# B&R Automation Studio project RS15_RX_30005_r00 (part 2)

#### Units.var
```iecst
(********************************************************************
 * COPYRIGHT --
 ********************************************************************
 * Program: Units
 * File: Units.var
 * Author: pkiel
 * Created: October 09, 2009
 ********************************************************************
 * Local variables of program Units
 ********************************************************************)
VAR RETAIN
	InchMetric_PB : BOOL;
END_VAR
```

### Program Logical/HMI/Language (IEC) - HMI Language Control

#### Language.var - Local variables
```iecst
(********************************************************************
 * COPYRIGHT --
 ********************************************************************
 * Program: Language
 * File: Language.var
 * Author: pkiel
 * Created: October 09, 2009
 ********************************************************************
 * Local variables of program Language
 ********************************************************************)
VAR RETAIN
	Language_PB : BOOL;
END_VAR
VAR
	Language_Ind : UINT;
END_VAR
```

### Program Logical/HMI/Password (IEC) - Password Control

#### PasswordCyclic.st
```iecst
(********************************************************************
 * COPYRIGHT --
 ********************************************************************
 * Program: Password
 * File: PasswordCyclic.st
 * Author: pkiel
 * Created: October 20, 2009
 ********************************************************************
 * Implementation of program Password
 ********************************************************************)

PROGRAM _CYCLIC

(* Evaluate Password...triggered from password completion bool on HMI *)
	IF (EvaluatePassword) THEN
		IF (PasswordEntered = gPassword.Supervisor) THEN
			UserLevel_Ind := 1;
		ELSE
			IF (PasswordEntered = gPassword.Maintenance) THEN
				UserLevel_Ind := 2;
			ELSE
				IF (PasswordEntered = gPassword.Technician) THEN
					UserLevel_Ind := 3;
				ELSE
					IF (PasswordEntered = '031168') THEN
						UserLevel_Ind := 3;
					ELSE
						InvalidPassword := 1;
						InvalidPassword_Ind := 0;
					END_IF
				END_IF
			END_IF
		END_IF
		PasswordEntered := '';
		EvaluatePassword := 0;
	END_IF

(* Invalid Password Indication *)
	TON_0(IN := InvalidPassword, PT := T#3s);
	IF (TON_0.Q) THEN
		InvalidPassword_Ind := 1;
		InvalidPassword := 0;
	END_IF

(* Logout Function...Forces User Level To "Operator" *)
	IF (Logout_PB) THEN
		UserLevel_Ind := 0;
		Logout_PB := 0;
	END_IF

(* Current User Indication *)
	CASE (UserLevel_Ind) OF
		0:
			DataLock_0 := 0;
			DataLock_1 := 2;
			DataLock_2 := 2;
			DataLock_3 := 2;
			CurrentUser := 'Operator';
		1:
			DataLock_0 := 0;
			DataLock_1 := 0;
			DataLock_2 := 2;
			DataLock_3 := 2;
			CurrentUser := 'Supervisor';
		2:
			DataLock_0 := 0;
			DataLock_1 := 0;
			DataLock_2 := 0;
			DataLock_3 := 2;
			CurrentUser := 'Maintenance';
		3:
			DataLock_0 := 0;
			DataLock_1 := 0;
			DataLock_2 := 0;
			DataLock_3 := 0;
			CurrentUser := 'Technician';
	END_CASE;

(* Detect Password Change Request *)
	IF (PasswordChangeStart_PB) THEN
		PasswordChange_Visibility := 0;
		PasswordChangeStart_PB := 0;
	END_IF

(* Password Change Validity Check *)
	IF (PasswordChangeAccept_PB) THEN
		IF (PasswordNew<>PasswordConfirm) THEN
			PasswordChangeFailure := 1;
			PasswordFail_Visibility := 0;
		ELSE
			StringLength := LEN(PasswordNew);
			IF (StringLength<5) THEN
				PasswordChangeFailure := 1;
				PasswordFail_Visibility := 0;
			ELSE
				IF(PasswordNew='00000') THEN
					PasswordChangeFailure := 1;
					PasswordFail_Visibility := 0;
				ELSE
					CASE (PasswordSelect_Ind) OF
						1:
							gPassword.Supervisor := PasswordNew;
						2:
							gPassword.Maintenance := PasswordNew;
						3:
							gPassword.Technician := PasswordNew;
					END_CASE
					PasswordChangeAccepted := 1;
					PasswordAccepted_Visibility := 0;
				END_IF
			END_IF
		END_IF
	PasswordChange_Visibility := 1;
	PasswordConfirm_Visibility :=1;
	PasswordNew := '';
	PasswordConfirm := '';
	PasswordSelect_Ind := 0;
	PasswordChangeAccept_PB := 0;
	END_IF

(* Password Change Accepted *)
	TON_1(IN := PasswordChangeAccepted, PT := T#3s);
	IF (TON_1.Q) THEN
		PasswordAccepted_Visibility := 1;
		PasswordChangeAccepted := 0;
	END_IF

(* Password Change Failure *)
	TON_2(IN := PasswordChangeFailure, PT := T#3s);
	IF (TON_2.Q) THEN
		PasswordFail_Visibility := 1;
		PasswordChangeFailure := 0;
	END_IF

(* Password Change Cancelled *)
	IF (PasswordChangeCancel_PB) THEN
		PasswordChange_Visibility := 1;
		PasswordConfirm_Visibility := 1;
		PasswordNew := '';
		PasswordConfirm := '';
		PasswordSelect_Ind := 0;
		PasswordChangeCancel_PB := 0;
	END_IF

  // Dryer Trend Button visibility
  IF (UserLevel_Ind > 1) THEN
    iDryerTrend_Visibility := 0 ; // Visible
  ELSE
    iDryerTrend_Visibility := 1 ;
  END_IF
END_PROGRAM
```

#### PasswordInit.st
```iecst
(********************************************************************
 * COPYRIGHT --
 ********************************************************************
 * Program: Password
 * File: PasswordInit.st
 * Author: pkiel
 * Created: October 20, 2009
 ********************************************************************
 * Implementation of program Password
 ********************************************************************)

PROGRAM _INIT

	UserLevel_Ind := 0;
	PasswordStatus := 0;
	InvalidPassword_Ind := 1;
	IF (NOT FirstBoot) THEN
		gPassword.Supervisor  := 'super';
		gPassword.Maintenance := 'maint';
		gPassword.Technician  := 'tech725';
		FirstBoot := 1;
	END_IF
	PasswordAccepted_Visibility := 1;
	PasswordChange_Visibility := 1;
	PasswordFail_Visibility := 1;
  PasswordConfirm_Visibility := 1;

  iDryerTrend_Visibility := 1 ;

END_PROGRAM
```

### Program Logical/HMI/Cmd_Trace (IEC) - Network Command Trace Transfer

#### Cmd_Trace.var
```iecst
(********************************************************************
 * COPYRIGHT --
 ********************************************************************
 * Program: Cmd_Trace
 * File: Cmd_Trace.var
 * Author: pkiel
 * Created: October 13, 2009
 ********************************************************************
 * Local variables of program Cmd_Trace
 ********************************************************************)
VAR
	MC_BR_NetTrace_0 : MC_BR_NetTrace;
	TraceErrorID : UINT;
	ErrorRecord : MC_ERRORRECORD_REF;
	Trace_PB : BOOL;
	TON_0 : TON;
	TON_1 : TON;
	TraceStatus : UINT;
	MessageTimer : BOOL;
END_VAR
```

#### Cmd_TraceCyclic.st
```iecst
(********************************************************************
 * COPYRIGHT --
 ********************************************************************
 * Program: Cmd_Trace
 * File: Cmd_TraceCyclic.st
 * Author: pkiel
 * Created: October 13, 2009
 ********************************************************************
 * Implementation of program Cmd_Trace
 ********************************************************************)

PROGRAM _CYCLIC

(* This program transfers the network command trace to a file named "Trace+Date" on a USB memory stick placed in the "USB1" location *)
	TON_0(IN:=Trace_PB,PT:=T#5s);

	IF (EDGEPOS(TON_0.Q)) THEN
		MC_BR_NetTrace_0.Execute:=TRUE;
		TraceStatus:=1;	(* Network Trace Transfer Started *)
	END_IF

	MC_BR_NetTrace_0.Command:=mcSAVE;
    MC_BR_NetTrace_0.Configuration.NetTrace.Type:=mcNET_TRACE_GLOBAL;
    strcpy(ADR(MC_BR_NetTrace_0.Configuration.DatObj.Name), ADR('Trace'));
    MC_BR_NetTrace_0.Configuration.DatObj.Type:=mcFILE + mcADD_DATE_TIME;
    strcpy(ADR(MC_BR_NetTrace_0.Configuration.DatObj.Device), ADR('USB1'));

    IF (MC_BR_NetTrace_0.Done) THEN
      MC_BR_NetTrace_0.Execute:=FALSE;
      TraceStatus:=2;	(* Network Trace Transfer Completed *)
    ELSIF (MC_BR_NetTrace_0.Error) THEN
      TraceErrorID:=MC_BR_NetTrace_0.ErrorID;
      ErrorRecord:=MC_BR_NetTrace_0.ErrorRecord;
      MC_BR_NetTrace_0.Execute:=FALSE;
      TraceStatus:=3;	(* Network Trace Transfer Error *)
    END_IF

    IF (TraceStatus=2 OR TraceStatus=3) THEN
    	MessageTimer:=1;
    ELSE
    	MessageTimer:=0;
    END_IF

    TON_1(IN:=MessageTimer,PT:=T#3s);
    IF EDGEPOS(TON_1.Q) THEN
    	TraceStatus:=0;
    END_IF

MC_BR_NetTrace_0();

END_PROGRAM
```

### Program Logical/HMI/Recipe_1 (IEC) - General Recipe Code

#### Recipe_1.var
```iecst
(********************************************************************
 * COPYRIGHT --
 ********************************************************************
 * Program: Recipe_1
 * File: Recipe_1.var
 * Author: pkiel
 * Created: October 13, 2009
 ********************************************************************
 * Local variables of program Recipe_1
 ********************************************************************)
VAR RETAIN
	RecipeCurrent_Index   : UINT;
  Repeat_Old            : REAL ;
  iAnimHoldTearEnvB_Old : INT ;
  iAnimHoldTearRS15_Old : INT ;
  rNumbPliers_Old       : REAL ;
END_VAR
VAR
	RecipeDropdown : UINT;
	RecipeLoad_PB : BOOL;
	RecipeSavePrompt : BOOL;
	RecipeSave_PB : BOOL;
	RecipeSaveAs_PB : BOOL;
	RecipeSelected : Recipe;
	RecipeDelete_PB : BOOL;
	ListBoxControl : UINT;
	RecipeViewSelect : UINT;
	RecipeLoadPopUp : UINT;
	RecipeSavePopUp : UINT;
	RecipeSaveAsPopUp : UINT;
	RecipeDeletePopUp : UINT;
	RecipeSavePromptText_Ind : UINT;
	RecipeSavePromptColor_Ind : UINT;
	RecipeSaveAsPopUp_PB : BOOL;
	RecipeTempName : STRING[32];
	TON_0 : TON;
  bNumPliersChange_Old : BOOL ;
  rRepeatMetric : REAL;
  rRepeatMetric_Old : REAL;
  iAnimHoldTearEnvB : INT ;
  iAnimHoldTearRS15 : INT ;
  iAnimDrum : INT ;
  rSP_PosRefEnvB : REAL ;
  HMI_rSPPosRefEnvB : REAL ;
  rHoldPerimeter_mm : REAL ;
  bResult : BOOL ;
  bAnimHoldTearEnvBChange : BOOL ;
  bAnimHoldTearRS15Change : BOOL ;
  rTempPosRefEnvB : REAL ;
END_VAR
```

#### Recipe_1Cyclic.st
```iecst
(********************************************************************
 * COPYRIGHT --
 ********************************************************************
 * Program: Recipe_1
 * File: Recipe_1Cyclic.st
 * Author: pkiel
 * Created: October 13, 2009
 ********************************************************************
 * Implementation of program Recipe_1
 ********************************************************************)

PROGRAM _CYCLIC

  RecipeDropdown := LIMIT (1,RecipeDropdown,50);
  RecipeSelected := gRecipeBase[RecipeDropdown];
  RecipeViewSelect := RecipeViewSelect;

  (* Recipe Load *)
  IF (RecipeLoad_PB) THEN
    gRecipeActive 				:= RecipeSelected;
    RecipeCurrent_Index 		:= RecipeDropdown;
    RecipeLoad_PB 				:= 0;
    gRecipeChange				:= 1;
    RecipeSavePrompt 			:= 0;
  END_IF

  (* Recipe Save *)
  IF (RecipeSave_PB) THEN
    gRecipeBase[RecipeCurrent_Index] := gRecipeActive;
    RecipeSavePrompt := 0;
    RecipeSave_PB :=0;
  END_IF

  ListBoxControl := ListBoxControl;

  (* Recipe Save As *)
  IF (RecipeSaveAsPopUp_PB) THEN
    RecipeTempName := gRecipeBase[RecipeDropdown].Name;
    RecipeSaveAsPopUp_PB := 0;
  END_IF
  IF (RecipeSaveAs_PB) THEN
    gRecipeBase[RecipeDropdown] := gRecipeActive;
    gRecipeBase[RecipeDropdown].Name := RecipeTempName;
    RecipeTempName:='';
    RecipeSavePrompt := 0;
    RecipeSaveAs_PB :=0;
  END_IF

  (* Recipe Delete *)
  IF (RecipeDelete_PB) THEN
    gRecipeBase[RecipeDropdown].Name 						       := 'BLANK RECIPE';
    gRecipeBase[RecipeDropdown].Repeat 						     := 0.0 ;
      gRecipeBase[RecipeDropdown].Drum_Offset			 		   := 0.0 ;
      gRecipeBase[RecipeDropdown].Entry_Draw					   := 0.0 ;
      gRecipeBase[RecipeDropdown].Exit_Draw					     := 0.0 ;
      gRecipeBase[RecipeDropdown].HoldCount					     := 0 ;
      gRecipeBase[RecipeDropdown].PackCount					     := 0 ;
      gRecipeBase[RecipeDropdown].Holding_Offset				 := 0.0 ;
      gRecipeBase[RecipeDropdown].Perf_Offset            := 0.0 ;
      gRecipeBase[RecipeDropdown].Tearing_Offset				 := 0.0 ;
      gRecipeBase[RecipeDropdown].rPerf_PhasMasterDeg    := 0.0 ;
      gRecipeBase[RecipeDropdown].rHolding_PhasMasterDeg := 0.0 ;
      gRecipeBase[RecipeDropdown].rTearing_PhasMasterDeg := 0.0 ;
      gRecipeBase[RecipeDropdown].rDrum_PhasMasterDeg    := 0.0 ;
      gRecipeBase[RecipeDropdown].bSelColdMicroPerfProd  := 0 ;
      gRecipeBase[RecipeDropdown].rCMPerf_PhasMasterDeg  := 0.0 ;
      gRecipeBase[RecipeDropdown].rCMPerf_Draw           := 0.0 ;
      gRecipeBase[RecipeDropdown].bCMPerf_Mode           := 0 ;
      gRecipeBase[RecipeDropdown].rHMPerf_PhasMasterDeg  := 0.0 ;
      gRecipeBase[RecipeDropdown].bHMPerf_Mode           := 0 ;
      gRecipeBase[RecipeDropdown].iHMPerf_Up             := 0 ;
      gRecipeBase[RecipeDropdown].rHotMicroPerfSize_in   := 0.0 ;
      gRecipeBase[RecipeDropdown].rTearEB_PhasMasterDeg  := 0.0 ;
      gRecipeBase[RecipeDropdown].bSelEnvBProd           := 0 ;
      gRecipeBase[RecipeDropdown].rEnvB_Offset           := 0.0 ;
      gRecipeBase[RecipeDropdown].rTearEB_Offset         := 0.0 ;
      gRecipeBase[RecipeDropdown].rEnvB_PerfSize_in      := 0.0 ;
      gRecipeBase[RecipeDropdown].rSlopeExitTable        := 0.0 ;
      gRecipeBase[RecipeDropdown].bSelTypeRSGlue         := 0 ;
      gRecipeBase[RecipeDropdown].bSelTypeOtherRSGlue    := 0 ;
      gRecipeBase[RecipeDropdown].bSelFPProd             := 0 ;
      gRecipeBase[RecipeDropdown].bSelHeaterProd         := 0 ;
      gRecipeBase[RecipeDropdown].rHeatSPDegF            := 0.0 ;
      gRecipeBase[RecipeDropdown].iNumToothGearPrint     := 0 ;
      gRecipeBase[RecipeDropdown].iPrintUp               := 0 ;
      RecipeDelete_PB :=0;
      END_IF

      (* Recipe Check: Is Current Recipe Changed From The Recipe That was Loaded? *)
      (*IF (RecipeCurrent.Name<>gRecipeBase[RecipeCurrent_Index].Name) THEN
      RecipeSavePrompt := 1;
      END_IF*)
      IF (gRecipeActive.Repeat <> gRecipeBase[RecipeCurrent_Index].Repeat) THEN
        RecipeSavePrompt := 1;
      END_IF
      IF (gRecipeActive.Drum_Offset <> gRecipeBase[RecipeCurrent_Index].Drum_Offset) THEN
        RecipeSavePrompt := 1;
      END_IF
      IF (gRecipeActive.Entry_Draw <> gRecipeBase[RecipeCurrent_Index].Entry_Draw) THEN
        RecipeSavePrompt := 1;
      END_IF
      IF (gRecipeActive.Exit_Draw <> gRecipeBase[RecipeCurrent_Index].Exit_Draw) THEN
        RecipeSavePrompt := 1;
      END_IF
      IF (gRecipeActive.HoldCount <> gRecipeBase[RecipeCurrent_Index].HoldCount) THEN
        RecipeSavePrompt := 1;
      END_IF
      IF (gRecipeActive.PackCount <> gRecipeBase[RecipeCurrent_Index].PackCount) THEN
        RecipeSavePrompt := 1;
      END_IF
      IF (gRecipeActive.Holding_Offset <> gRecipeBase[RecipeCurrent_Index].Holding_Offset) THEN
        RecipeSavePrompt := 1;
      END_IF
      IF (gRecipeActive.Perf_Offset <> gRecipeBase[RecipeCurrent_Index].Perf_Offset) THEN
        RecipeSavePrompt := 1;
      END_IF
      IF (gRecipeActive.Tearing_Offset <> gRecipeBase[RecipeCurrent_Index].Tearing_Offset) THEN
        RecipeSavePrompt := 1;
      END_IF
      IF (gRecipeActive.rPerf_PhasMasterDeg <> gRecipeBase[RecipeCurrent_Index].rPerf_PhasMasterDeg) THEN
        RecipeSavePrompt := 1;
      END_IF
      IF (gRecipeActive.rHolding_PhasMasterDeg <> gRecipeBase[RecipeCurrent_Index].rHolding_PhasMasterDeg) THEN
        RecipeSavePrompt := 1;
      END_IF
      IF (gRecipeActive.rTearing_PhasMasterDeg <> gRecipeBase[RecipeCurrent_Index].rTearing_PhasMasterDeg) THEN
        RecipeSavePrompt := 1;
      END_IF
      IF (gRecipeActive.rDrum_PhasMasterDeg <> gRecipeBase[RecipeCurrent_Index].rDrum_PhasMasterDeg) THEN
        RecipeSavePrompt := 1;
      END_IF
      IF (gRecipeActive.rCMPerf_OffsetIn <> gRecipeBase[RecipeCurrent_Index].rCMPerf_OffsetIn) THEN
        RecipeSavePrompt := 1;
      END_IF
      IF (gRecipeActive.rCMPerf_PhasMasterDeg <> gRecipeBase[RecipeCurrent_Index].rCMPerf_PhasMasterDeg) THEN
        RecipeSavePrompt := 1;
      END_IF
      IF (gRecipeActive.rHMPerf_OffsetIn <> gRecipeBase[RecipeCurrent_Index].rHMPerf_OffsetIn) THEN
        RecipeSavePrompt := 1;
      END_IF
      IF (gRecipeActive.rHMPerf_PhasMasterDeg <> gRecipeBase[RecipeCurrent_Index].rHMPerf_PhasMasterDeg) THEN
        RecipeSavePrompt := 1;
      END_IF
      IF (gRecipeActive.rCMPerf_Draw <> gRecipeBase[RecipeCurrent_Index].rCMPerf_Draw) THEN
        RecipeSavePrompt := 1;
      END_IF
      IF (gRecipeActive.rHotMicroPerfSize_in <> gRecipeBase[RecipeCurrent_Index].rHotMicroPerfSize_in) THEN
        RecipeSavePrompt := 1;
      END_IF
      IF (gRecipeActive.bSelFPProd <> gRecipeBase[RecipeCurrent_Index].bSelFPProd) THEN
        RecipeSavePrompt := 1;
      END_IF
      IF (gRecipeActive.bSelHeaterProd <> gRecipeBase[RecipeCurrent_Index].bSelHeaterProd) THEN
        RecipeSavePrompt := 1;
      END_IF
      IF (gRecipeActive.rHeatSPDegF <> gRecipeBase[RecipeCurrent_Index].rHeatSPDegF) THEN
        RecipeSavePrompt := 1 ;
      END_IF
      IF (gRecipeActive.bSelColdMicroPerfProd <> gRecipeBase[RecipeCurrent_Index].bSelColdMicroPerfProd) THEN
        RecipeSavePrompt := 1;
      END_IF
      IF (gRecipeActive.rSlopeExitTable <> gRecipeBase[RecipeCurrent_Index].rSlopeExitTable) THEN
        RecipeSavePrompt := 1;
      END_IF
      IF (gRecipeActive.bSelTypeRSGlue <> gRecipeBase[RecipeCurrent_Index].bSelTypeRSGlue) THEN
        RecipeSavePrompt := 1;
      END_IF
      IF (gRecipeActive.iNumToothGearPrint <> gRecipeBase[RecipeCurrent_Index].iNumToothGearPrint) THEN
        RecipeSavePrompt := 1;
      END_IF
      IF (gRecipeActive.iPrintUp <> gRecipeBase[RecipeCurrent_Index].iPrintUp) THEN
        RecipeSavePrompt := 1;
      END_IF
      IF (gRecipeActive.rEnvB_PhasMasterDeg <> gRecipeBase[RecipeCurrent_Index].rEnvB_PhasMasterDeg) THEN
        RecipeSavePrompt := 1;
      END_IF
      IF (gRecipeActive.rTearEB_PhasMasterDeg <> gRecipeBase[RecipeCurrent_Index].rTearEB_PhasMasterDeg) THEN
        RecipeSavePrompt := 1;
      END_IF
      IF (gRecipeActive.rEnvB_Offset <> gRecipeBase[RecipeCurrent_Index].rEnvB_Offset) THEN
        RecipeSavePrompt := 1;
      END_IF
      IF (gRecipeActive.rTearEB_Offset <> gRecipeBase[RecipeCurrent_Index].rTearEB_Offset) THEN
        RecipeSavePrompt := 1;
      END_IF
      IF (gRecipeActive.rEnvB_PerfSize_in <> gRecipeBase[RecipeCurrent_Index].rEnvB_PerfSize_in) THEN
        RecipeSavePrompt := 1;
      END_IF
      IF (gRecipeActive.rHMPerf_PhasMasterDeg <> gRecipeBase[RecipeCurrent_Index].rHMPerf_PhasMasterDeg) THEN
        RecipeSavePrompt := 1;
      END_IF
      IF (gRecipeActive.bCMPerf_Mode <> gRecipeBase[RecipeCurrent_Index].bCMPerf_Mode) THEN
        RecipeSavePrompt := 1;
      END_IF
      IF (gRecipeActive.bHMPerf_Mode <> gRecipeBase[RecipeCurrent_Index].bHMPerf_Mode) THEN
        RecipeSavePrompt := 1;
      END_IF
      IF (gRecipeActive.iHMPerf_Up <> gRecipeBase[RecipeCurrent_Index].iHMPerf_Up) THEN
        RecipeSavePrompt := 1;
      END_IF
      IF (gRecipeActive.bSelEnvBProd <> gRecipeBase[RecipeCurrent_Index].bSelEnvBProd) THEN
        RecipeSavePrompt := 1;
      END_IF
      IF (gRecipeActive.bSelTypeOtherRSGlue <> gRecipeBase[RecipeCurrent_Index].bSelTypeOtherRSGlue) THEN
        RecipeSavePrompt := 1;
      END_IF

      IF (RecipeSavePrompt) THEN
        RecipeSavePromptText_Ind := 1;
        RecipeSavePromptColor_Ind := gRed+(256*gBlack);
      ELSE
        RecipeSavePromptText_Ind := 0;
        RecipeSavePromptColor_Ind := 34+(256*gBlack);
      END_IF

      IF g_bSplashDone THEN
        // Detect Number pliers on Drum Change
        rRepeatMetric := gRecipeActive.Repeat*25.4;
          rRepeatMetric_Old := Repeat_Old*25.4;

          (* Detect Repeat Change *)
          IF ((gRecipeActive.Repeat<>Repeat_Old)OR (gRecipeChange)) THEN
            gRepeatChange:=1;
            gRecipeChange:=0;
            Repeat_Old := gRecipeActive.Repeat;
              END_IF
              // Number of pliers on Drum calc
              IF (rRepeatMetric > gr_rBagSize4_2Pliers_mm) OR
                gRecipeActive.bSelEnvBProd                THEN
                g_rNumbPliers := 2.0 ;
              ELSE
                g_rNumbPliers := 4.0 ;
              END_IF ;
              // Detect number of pliers change on Drum
              IF (g_rNumbPliers <> rNumbPliers_Old) THEN
                g_bNumPliersChange := 1 ;
                rNumbPliers_Old := g_rNumbPliers;
                // Detect change from 4 to 2 pliers on Drum
                IF (rRepeatMetric > gr_rBagSize4_2Pliers_mm)      AND
                  (rRepeatMetric_Old <= gr_rBagSize4_2Pliers_mm) THEN
                  g_bNumPliersChange4to2[1] := 1 ;
                  g_bNumPliersChange4to2[2] := 1 ;
                ELSE
                  // Detect change from 2 to 4 pliers on Drum
                  g_bNumPliersChange2to4[1] := 1 ;
                END_IF
              END_IF
              IF g_bNumPliersChange4to2[1] OR
                g_bNumPliersChange2to4[1] THEN
                // Change Modulo on Tearing and Drum
                g_bChangeModTearingReq := 1 ;
                g_bChangeModDrumReq    := 1 ;
                g_bChangeModTearEBReq  := 1 ;
              END_IF

              // Drum picture animation
              IF g_iMachType <> C_iRS15 THEN
                iAnimDrum := REAL_TO_INT(g_rNumbPliers) ;
              ELSE
                iAnimDrum := 5 ;
              END_IF

              // Number of maintaining case RS15
              IF (rRepeatMetric>=gr_rBagSize2_4Hold_mm) THEN
                iAnimHoldTearRS15 := 2 ;
              ELSE
                iAnimHoldTearRS15 := 4 ;
              END_IF

              TON_0( IN:=gRepeatChange, PT:=T#1s );
              IF (TON_0.Q) THEN
                gRepeatChange      := 0 ;
                g_bNumPliersChange := 0 ;
              END_IF
              // Display screen config HoldTearDrum
              gHMI_GoToHoldTearDrum_PB := EDGEPOS(g_bNumPliersChange) OR EDGEPOS(bAnimHoldTearEnvBChange) OR EDGEPOS(bAnimHoldTearRS15Change) ;
              // Indicator Tearing on the first station
              gr_rIndEnvB2AxTear1 := 0 ;

              IF gA[13].bInMach THEN  // Case Envelope Bag 2 Axis
                rHoldPerimeter_mm := gr_rBagSize2_4Hold_mm*2.0 ;
                IF gRecipeActive.bSelEnvBProd THEN
                  IF (rRepeatMetric<=rHoldPerimeter_mm) THEN
                    iAnimHoldTearEnvB := 4 ;
                  ELSE
                    iAnimHoldTearEnvB := 5 ;
                  END_IF
                  rSP_PosRefEnvB := gr_rPosEnvBHoldBag ;
                ELSE
                  IF (g_rNumbPliers=4) THEN
                    iAnimHoldTearEnvB := 1 ;
                  ELSIF (g_rNumbPliers=2)                       AND
                    (rRepeatMetric<=gr_rEnvBSizeTear2_1_mm) THEN
                    gr_rIndEnvB2AxTear1 := 0 ; // Indicator Tearing on the first station
                    iAnimHoldTearEnvB := 2 ;
                  ELSE
                    gr_rIndEnvB2AxTear1 := 1 ; // Indicator Tearing on the first station
                    iAnimHoldTearEnvB := 3 ;
                  END_IF
                  rTempPosRefEnvB := gr_rPosEnvBHoldBag + 45.0 ;
                  rSP_PosRefEnvB := H_FC_Modulus (
                    IN_rMod := 360.0 ,
                    IN_rVar := rTempPosRefEnvB
                    ) ;
                END_IF
              END_IF
              g_EnvB_iHoldTearEnvBCase := iAnimHoldTearEnvB ;
              bAnimHoldTearEnvBChange := (iAnimHoldTearEnvB_Old<>iAnimHoldTearEnvB) ;
              bAnimHoldTearRS15Change := (iAnimHoldTearRS15_Old<>iAnimHoldTearRS15) ;
              iAnimHoldTearEnvB_Old := iAnimHoldTearEnvB ;
              iAnimHoldTearRS15_Old := iAnimHoldTearRS15 ;
              HMI_rSPPosRefEnvB := rSP_PosRefEnvB ;
              END_IF

              END_PROGRAM
```

#### Recipe_1Init.st
```iecst
(********************************************************************
 * COPYRIGHT --
 ********************************************************************
 * Program: Recipe_1
 * File: Recipe_1Init.st
 * Author: pkiel
 * Created: October 13, 2009
 ********************************************************************
 * Implementation of program Recipe_1
 ********************************************************************)

PROGRAM _INIT

	RecipeLoadPopUp := 1;
	RecipeSavePopUp := 1;
	RecipeSaveAsPopUp := 1;
	RecipeDeletePopUp := 1;
	RecipeCurrent_Index := LIMIT(1,RecipeCurrent_Index,50);

END_PROGRAM
```

### Program Logical/HMI/Recipe_2 (IEC) - Recipe Backup & Restore

#### Recipe_2Cyclic.st
```iecst
(********************************************************************
 * COPYRIGHT --
 ********************************************************************
 * Program: Recipe_2
 * File: Recipe_2Cyclic.st
 * Author: pkiel
 * Created: November 16, 2009
 ********************************************************************
 * Implementation of program Recipe_2
 ********************************************************************)

PROGRAM _CYCLIC

strcpy(ADR(gRecipeCntl.currRecipe), ADR(recipeName[indexNum]));

CASE step OF

	INIT_WAIT:
		IF(waitCnt > 100)THEN
			waitCnt 	:= 0;
			step 		:= INIT_RECIPE;
		ELSE
			waitCnt := waitCnt + 1;
		END_IF

	INIT_RECIPE:
		(**** Get directory info ****)
		(* Initialize info structure *)

		DirInfo_0(enable:=1, pDevice:= pDevice[gRecipeCntl.driveSelect], pPath:=ADR(''));

		(* Get FBK output information *)
		dirNum		:= DirInfo_0.dirnum;
		fileNum 	:= DirInfo_0.filenum;

		                           		  (*01234567890123456789*)
		strcpy(ADR(gRecipeCntl.status),ADR('READ DIR INFO'));

		(* Verify status *)
		IF (DirInfo_0.status = 0) THEN
			step := INIT_RECIPE + 1;
			(* Verify number of files found *)
			IF (fileNum >= MAX_RECIPE) THEN
				fileNum := MAX_RECIPE;
			END_IF
			fileCounter := 0;
			memset(ADR(readDir),0,SIZEOF(readDir));
			memset(ADR(recipeName),0,SIZEOF(recipeName));
			memset(ADR(recipeDescription),0,SIZEOF(recipeDescription));

			driveSelectOld	:= gRecipeCntl.driveSelect;

		ELSE
			IF (DirInfo_0.status <> 65535) THEN

				IF(DirInfo_0.status = fiERR_FILE_DEVICE)THEN

					IF(gRecipeCntl.driveSelect < 2)THEN
						gRecipeCntl.driveSelect := gRecipeCntl.driveSelect + 1;
					ELSE
														  (*01234567890123456789*)
						strcpy(ADR(gRecipeCntl.status),ADR('USB NOT CONNECTED'));
						gRecipeCntl.driveSelect := driveSelectOld;

						step 	:= COMMAND_RECIPE;
						stsCnt 	:= 0;

					END_IF

				ELSE
					errorLevel		:= 2;
					errStep 		:= step;
					step 			:= ERROR_STEP;

					IF (DirInfo_0.status = 20799) THEN
						wError := FileIoGetSysError();
					ELSE
						wError := DirInfo_0.status;
					END_IF
				END_IF

			END_IF
		END_IF

	11:

		(**** Get directory info ****)
		(* Verify counter variable *)
		IF (fileCounter < fileNum) THEN
			(* Initialize read directory structure *)
			DirRead_0(enable:= 1, pDevice:= DirInfo_0.pDevice, pPath:= 0, entry:= fileCounter, option:= FILE_FILE, pData:= ADR(readDir), data_len:= SIZEOF(readDir));

			itoa((fileCounter + 1), ADR(countString));
			itoa(fileNum, ADR(totalNumString));

									  		  (*01234567890123456789*)
			strcpy(ADR(gRecipeCntl.status),ADR('READ FILE '));
			strcat(ADR(gRecipeCntl.status),ADR(countString));
			strcat(ADR(gRecipeCntl.status),ADR(' OF '));
			strcat(ADR(gRecipeCntl.status),ADR(totalNumString));

			(* Verify status *)
			IF (DirRead_0.status = 0) THEN
				step 	:= INIT_RECIPE + 2;

			ELSE
				IF (DirRead_0.status <> 65535) THEN
					errorLevel		:= 3;
					errStep 		:= step;
					step 			:= ERROR_STEP;

					IF (DirRead_0.status = 20799) THEN
						wError := FileIoGetSysError();
					ELSE
						wError := DirRead_0.status;
					END_IF
				END_IF
			END_IF

		ELSE
			step 	:= COMMAND_RECIPE;
			stsCnt 	:= 0;

		END_IF

	12:
		(**** Try to open existing file ****)
		(* Initialize file open structrue *)
		FileOpen_0(enable:=1, pDevice:=DirInfo_0.pDevice, pFile:= ADR(readDir.Filename), mode:=FILE_R);

			 					   		  (*01234567890123456789*)
		(*strcpy(ADR(gRecipeCntl.status),ADR('OPEN RECIPE FILE'));*)

		(* Verify status (20708 -> File doesn't exist) *)
		IF (FileOpen_0.status = 20708) THEN
			step 		:= INIT_RECIPE + 1;
			fileCounter := fileCounter + 1;
		ELSE
			IF (FileOpen_0.status = 0) THEN
				memset(ADR(recipeDescriptionTemp),0,SIZEOF(recipeDescriptionTemp));
				step := INIT_RECIPE + 3;
			ELSE
				IF (FileOpen_0.status <> 65535) THEN
					errorLevel		:= 4;
					errStep 		:= step;
					step 			:= ERROR_STEP;

					IF (FileOpen_0.status = 20799) THEN
						wError := FileIoGetSysError();
					ELSE
						wError := FileOpen_0.status;
					END_IF
				END_IF
			END_IF
		END_IF

	13:
		(**** Read data from file - description****)
		(* Initialize file read structure *)

		FileRead_0(enable:=1, ident:=FileOpen_0.ident, offset:=114, pDest:= ADR(recipeDescriptionTemp), len:=SIZEOF(recipeDescription[fileCounter]));

			 					   		  (*01234567890123456789*)
		(*strcpy(ADR(gRecipeCntl.status),ADR('READ DESCRIPTION'));*)

		(* Verify status *)
		IF (FileRead_0.status = 0) THEN
			step := INIT_RECIPE + 4;
			strLenChk := strlen(ADR(readDir.Filename));

			IF(strLenChk > 4)THEN

				memChk := memcmp((ADR(readDir.Filename) + strLenChk - 4),ADR('.CSV') , 4);

				IF(memChk = 0)THEN
					(*Copy the name of the file*)
					memcpy(ADR(recipeName[fileCounter]),ADR(readDir.Filename), (strLenChk));

					(*Copy the recipe description*)
					FOR cnt := 0 TO 79 DO

						pChar ACCESS ADR(recipeDescriptionTemp) + cnt;
						IF(pChar = CR)THEN
							EXIT;
						END_IF
					END_FOR
					memcpy(ADR(recipeDescription[fileCounter]),ADR(recipeDescriptionTemp),cnt);
				END_IF

			END_IF

			fileCounter := fileCounter + 1;
		ELSE
			IF (FileRead_0.status <> 65535) THEN
				errorLevel		:= 5;
				errStep 		:= step;
				step 			:= ERROR_STEP;

				IF (FileRead_0.status = 20799) THEN
					wError := FileIoGetSysError();
				ELSE
					wError := FileRead_0.status;
				END_IF
			END_IF

		END_IF

	14:
		(**** Close the file ****)
		(* Initialize file close structure *)
		FileClose_0(enable:=1, ident:=FileOpen_0.ident);

			 					   		  (*01234567890123456789*)
		(*strcpy(ADR(gRecipeCntl.status),ADR('CLOSE FILE'));*)

		(* Verify status *)
   		IF (FileClose_0.status = 0) THEN
 			step := INIT_RECIPE + 1;
   		ELSE
			IF (FileClose_0.status <> 65535) THEN
				errorLevel		:= 6;
				errStep 		:= step;
				step 			:= ERROR_STEP;

				IF (FileClose_0.status = 20799) THEN
					wError := FileIoGetSysError();
				ELSE
					wError := FileClose_0.status;
				END_IF
			END_IF

		END_IF

	COMMAND_RECIPE:

		IF(stsCnt > 200)THEN
			gRecipeCntl.opActive := 0;
					  				      	  (*012345678901234567890123456789*)
			strcpy(ADR(gRecipeCntl.status),ADR('READY'));
		ELSE
			stsCnt := stsCnt + 1;
		END_IF

		IF(gRecipeCntl.cmdDelete)THEN
			gRecipeCntl.cmdDelete  	:= 0;
			gRecipeCntl.opActive 	:= 1;
			step := DELETE_RECIPE;

		ELSIF(gRecipeCntl.cmdLoad)THEN

			gRecipeCntl.cmdLoad		:= 0;
			gRecipeCntl.opActive 	:= 1;
			step := LOAD_RECIPE;

		ELSIF(gRecipeCntl.cmdSave) THEN

			gRecipeCntl.cmdSave 	:= 0;
			gRecipeCntl.opActive 	:= 1;
			step := SAVE_RECIPE;
		ELSIF(driveSelectOld <> gRecipeCntl.driveSelect)THEN
			step := INIT_RECIPE;
		END_IF

	DELETE_RECIPE:

		(**** Delete the file ****)
		(* Initialize file delete structure *)
		strcpy(ADR(tempString),ADR(gRecipeCntl.currRecipe));
		(*strcat(ADR(tempString),ADR('.CSV'));*)

		FileDelete_0(enable:=1, pDevice:=pDevice[gRecipeCntl.driveSelect], pName:=ADR(tempString));

			 					   		  (*01234567890123456789*)
		strcpy(ADR(gRecipeCntl.status),ADR('DELETE FILE'));

		(* Verify status *)
   		IF ((FileDelete_0.status = 0) OR (FileDelete_0.status = fiERR_FILE_NOT_FOUND)) THEN
 			step := INIT_WAIT;
   		ELSE
			IF (FileDelete_0.status <> 65535) THEN
				errorLevel		:= 10;
				errStep 		:= step;
				step 			:= ERROR_STEP;

				IF (FileDelete_0.status = 20799) THEN
					wError := FileIoGetSysError();
				ELSE
					wError := FileDelete_0.status;
				END_IF
			END_IF

		END_IF

	SAVE_RECIPE:
		(*IF(strlen(ADR(gRecipeCntl.newRecipe)) > 0)THEN*)
			(****      Create CSV file     ****)
			(*   Initialize file CSV search   *)

			CSV_Search_0(pStructName:=ADR(pNames), NumOfStructs:=1, pStructMem:=CSV_Init_0.pStructMem, MemLen:=CSV_Init_0.MemCounter,
			Options:=0, FullNameLenght:= CSV_Init_0.FullNameLenght, FileHeader:=1, Separator:= 59, pMaschineNo:=0, pComment:=ADR('Recipe Backup File'), pVersion:=0);

											  (*01234567890123456789*)
			strcpy(ADR(gRecipeCntl.status),ADR('CREATING CSV FILE'));

			(* Verify status *)
	   		IF (CSV_Search_0.status = 0) THEN
	 			step := SAVE_RECIPE + 1;
	   		ELSE
				IF (CSV_Search_0.status <> 65535) THEN
					errorLevel		:= 10;
					errStep 		:= step;
					step 			:= ERROR_STEP;

					IF (CSV_Search_0.status = 20799) THEN
						wError := FileIoGetSysError();
					ELSE
						wError := CSV_Search_0.status;
					END_IF
				END_IF

			END_IF

		(*ELSE
										      (*01234567890123456789*)
			(*strcpy(ADR(gRecipeCntl.status),ADR('NO RECIPE NAME'));
			step := ERROR_STEP;
		END_IF*)

	71:
		(**** Write CSV file            ****)
		(* Initialize file write structrue *)
		strcpy(ADR(tempString),ADR('Recipe'));

		CSV_WriteFile_0(pFileName:=ADR(tempString), pDevice:=pDevice[gRecipeCntl.driveSelect], pStructMem:=CSV_Init_0.pStructMem,
       	MemLen:= CSV_Search_0.FileLen, Mode:= FILE_OW);

		   	 					   	  	  (*01234567890123456789*)
		strcpy(ADR(gRecipeCntl.status),ADR('SAVING TO CSV FILE'));

		IF (CSV_WriteFile_0.status = 0) THEN
			step := INIT_WAIT;
		ELSE
			IF (CSV_WriteFile_0.status <> 65535) THEN
				errorLevel		:= 10;
				errStep 		:= step;
				step 			:= ERROR_STEP;

				IF (CSV_WriteFile_0.status = 20799) THEN
					wError := FileIoGetSysError();
				ELSE
					wError := CSV_WriteFile_0.status;
				END_IF
			END_IF
		END_IF

	LOAD_RECIPE:
		(**** Read CSV file 	      ****)
		(* Initialize Read CSV structrue *)
		strcpy(ADR(tempString),ADR('Recipe'));

		CSV_ReadFile_0(pFileName:=ADR(tempString), pDevice:=pDevice[gRecipeCntl.driveSelect], No_DatatypControl:=0, Separator:=59, Options:=0);

			 					   	      (*01234567890123456789*)
		strcpy(ADR(gRecipeCntl.status),ADR('LOADING DATA FROM CSV FILE'));

		IF (CSV_ReadFile_0.status = 0) THEN
			step := INIT_WAIT;
		ELSE
			IF (CSV_ReadFile_0.status <> 65535) THEN
				errorLevel		:= 20;
				errStep 		:= step;
				step 			:= ERROR_STEP;

				IF (CSV_ReadFile_0.status = 20799) THEN
					wError := FileIoGetSysError();
				ELSE
					wError := CSV_ReadFile_0.status;
				END_IF
			END_IF
		END_IF

	ERROR_STEP:
									   (*01234567890123456789*)
		strcpy(ADR(gRecipeCntl.status),ADR('ERROR NUM-'));
		itoa(wError, ADR(errorString));
		strcat(ADR(gRecipeCntl.status),ADR(errorString));
		step 	:= INIT_WAIT;

END_CASE

IF(gRecipeCntl.driveSelect = 0)THEN
	hmiDevice := 0;
END_IF

END_PROGRAM
```

#### Recipe_2Init.st
```iecst
(********************************************************************
 * COPYRIGHT --
 ********************************************************************
 * Program: Recipe_2
 * File: Recipe_2Init.st
 * Author: pkiel
 * Created: November 16, 2009
 ********************************************************************
 * Implementation of program Recipe_2
 ********************************************************************)

PROGRAM _INIT

(*Name of the recipe data structure*)
	pNames[0]:=ADR('gRecipeBase');

	CSV_Init_0(pStructName:=ADR(pNames), NumOfStructs:=1, FullNameLenght:=0, Options:=0);

(*Setup hardware axis as defined in the CPU->properties->file device*)
	(*pDevice[0]	:= ADR('RECIPE');*)
	pDevice[1]	:= ADR('USB1');
	pDevice[2]	:= ADR('USB2');

	step 		:= INIT_WAIT;
	indexNum	:= 0;
	hmiDevice	:= 1;

	gRecipeCntl.cmdDelete	:= FALSE;
	gRecipeCntl.cmdLoad		:= FALSE;
	gRecipeCntl.cmdSave		:= FALSE;
	gRecipeCntl.driveSelect := 1;
	RecipeBackUpPopUp := 1;
	RecipeRestorePopUp := 1;

END_PROGRAM
```

### Program Logical/HMI/Message_1 (IEC) - Message Display #1 Code

#### Message_1.var
```iecst
(********************************************************************
 * COPYRIGHT --
 ********************************************************************
 * Program: Message_1
 * File: Message_1.var
 * Author: pkiel
 * Created: October 16, 2009
 ********************************************************************
 * Local variables of program Message_1
 ********************************************************************)
VAR
	FirstMessage_L1 : BOOL;
	FirstMessage_L2 : BOOL;
	HGW_2StateIND_0 : HGW_2StateIND;
	HMI_MessageDisplay : UINT;
	Message : ARRAY[0..100] OF BOOL;
	MessageActive : BOOL;
	MessageColor_Ind : UINT;
	MessageDisplay : UINT;
	MessageReset : BOOL;
	MessageStatus : UINT;
	Permissive_L2 : BOOL;
	Permissive_L3 : BOOL;
	SelfReset : BOOL;
	SparePermissive : BOOL;
	TON_0 : TON;
END_VAR
```

#### Message_1Cyclic.ld
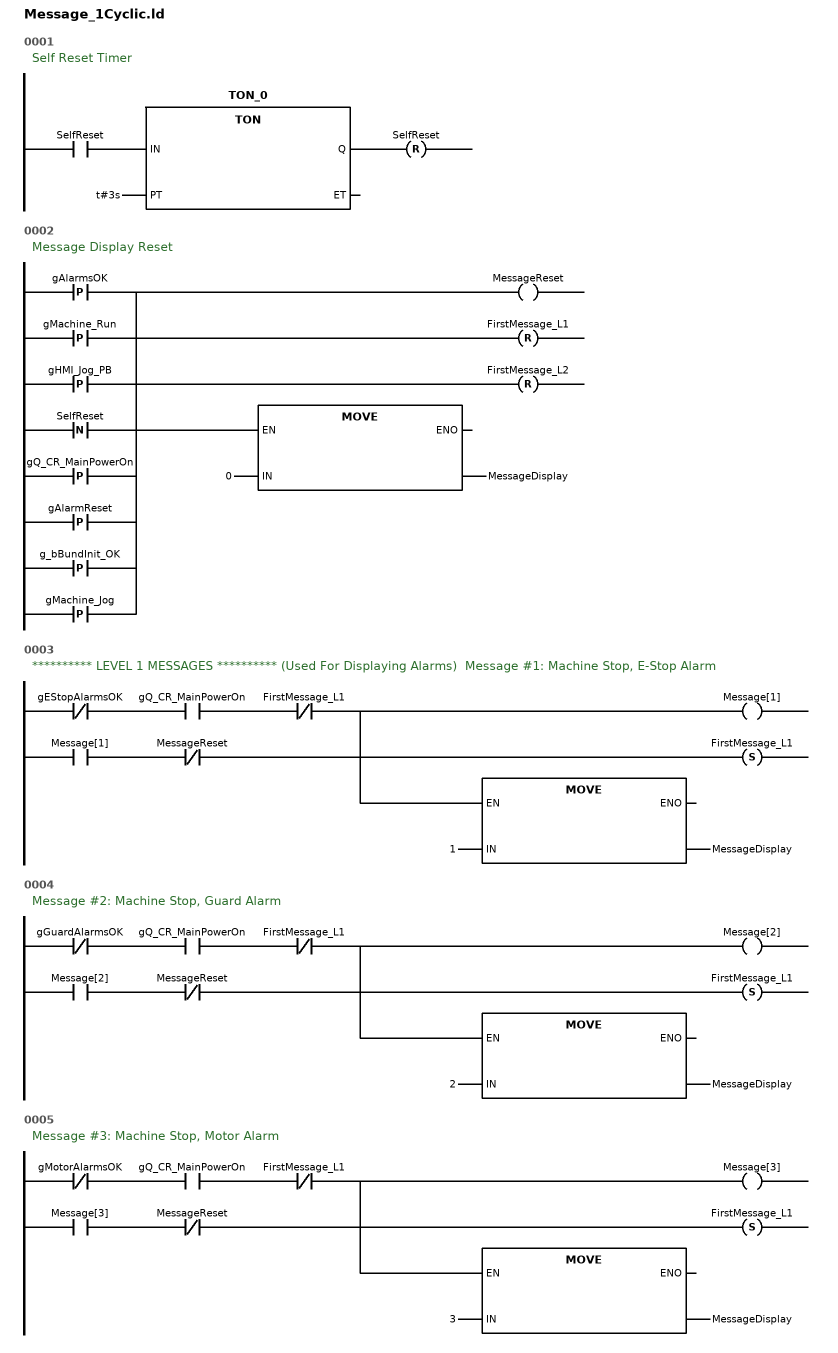
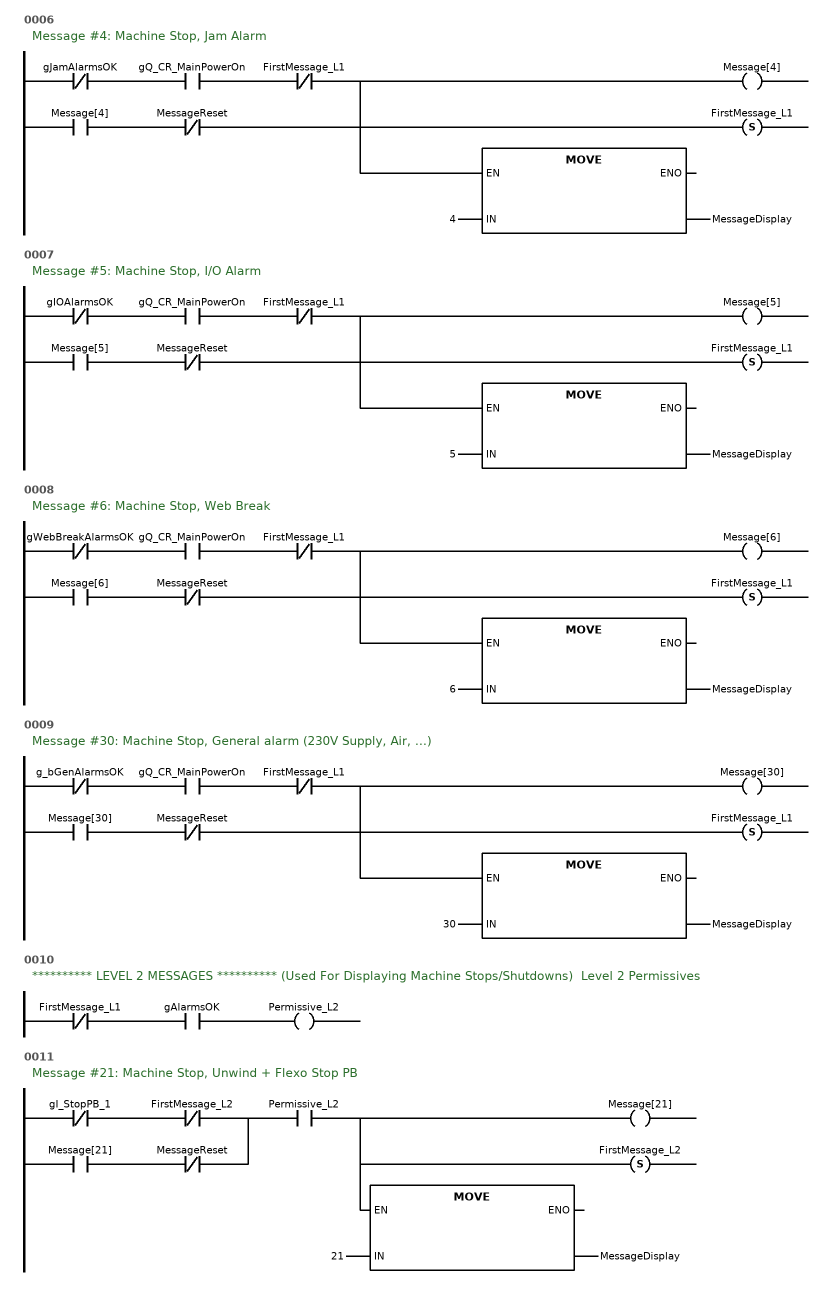
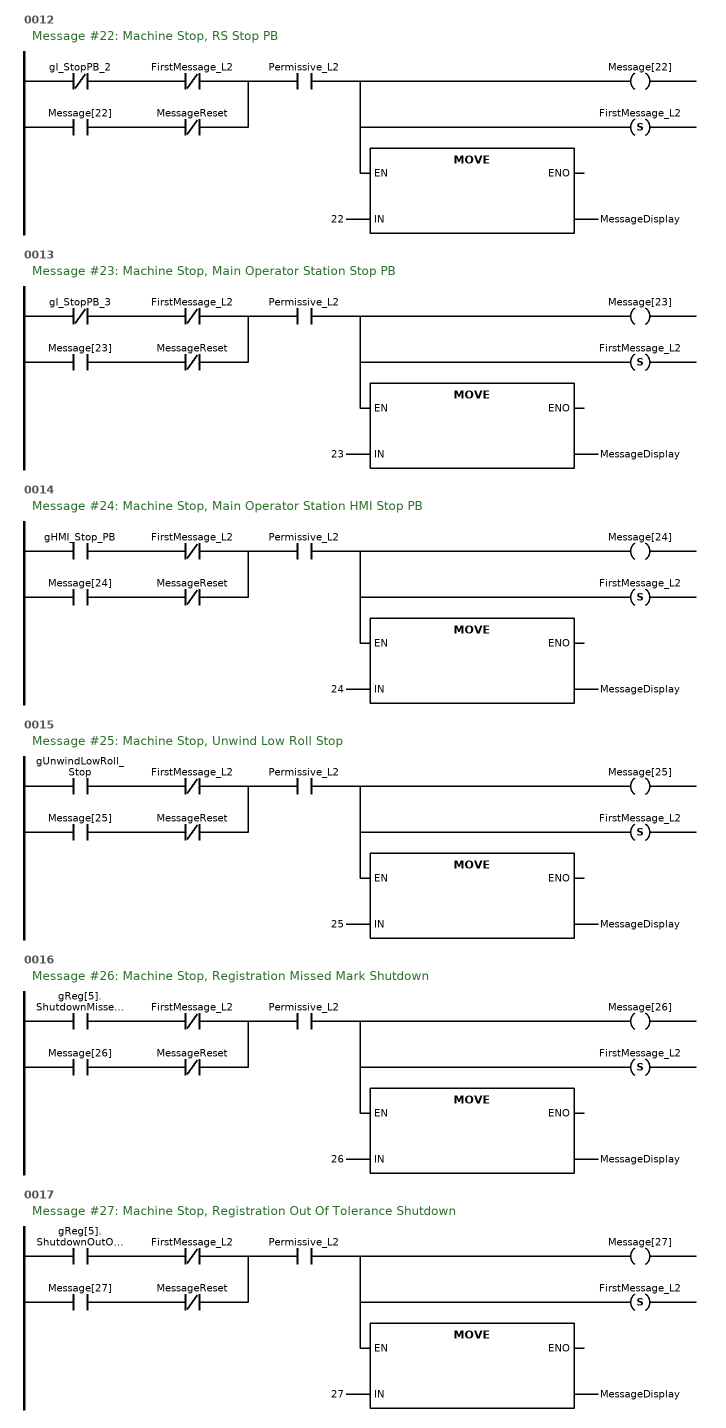
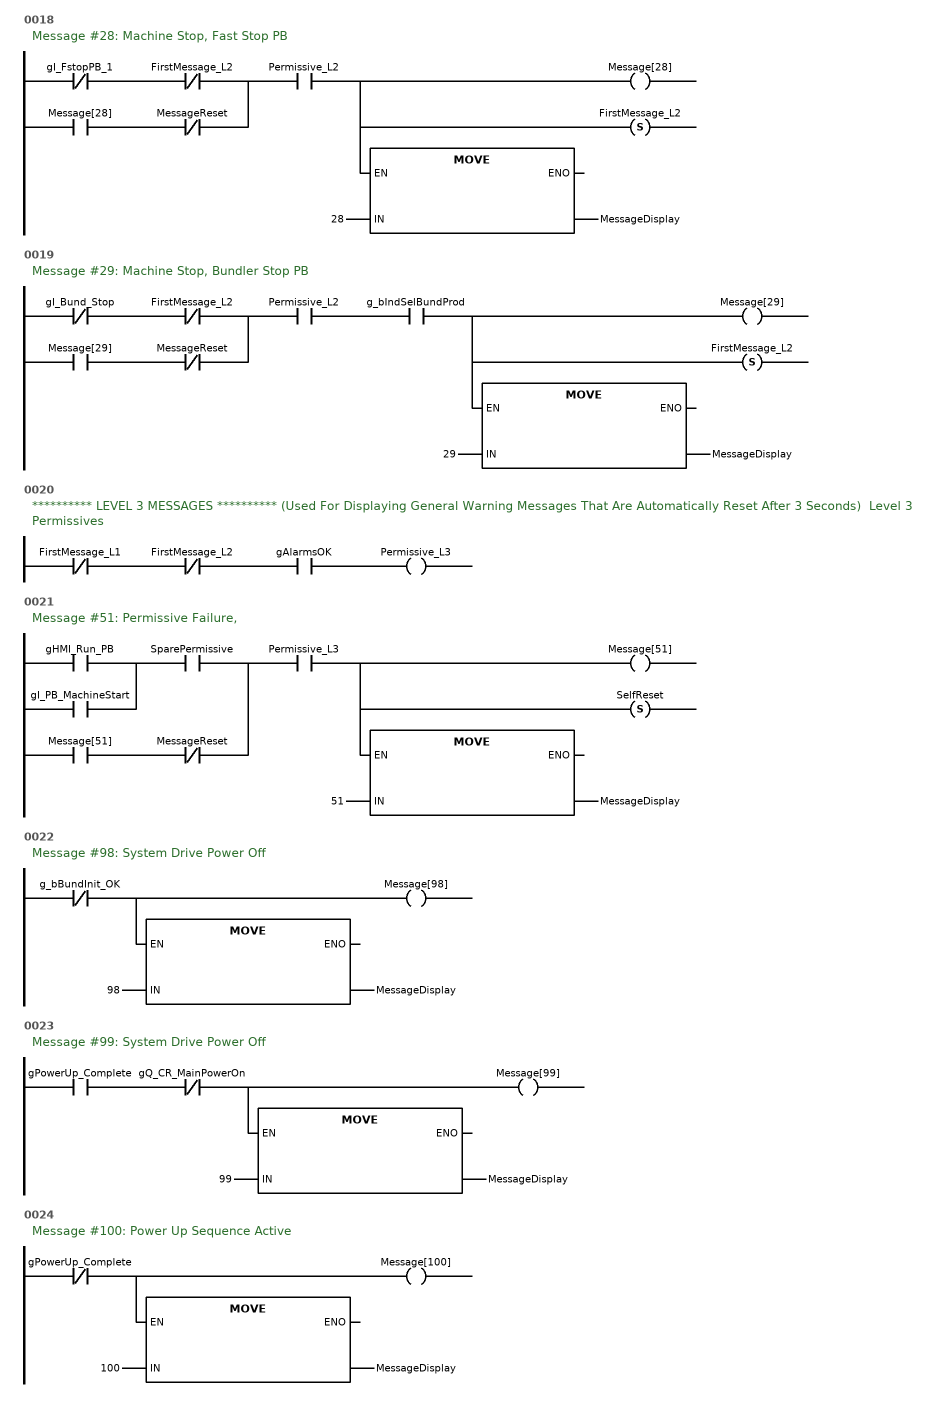
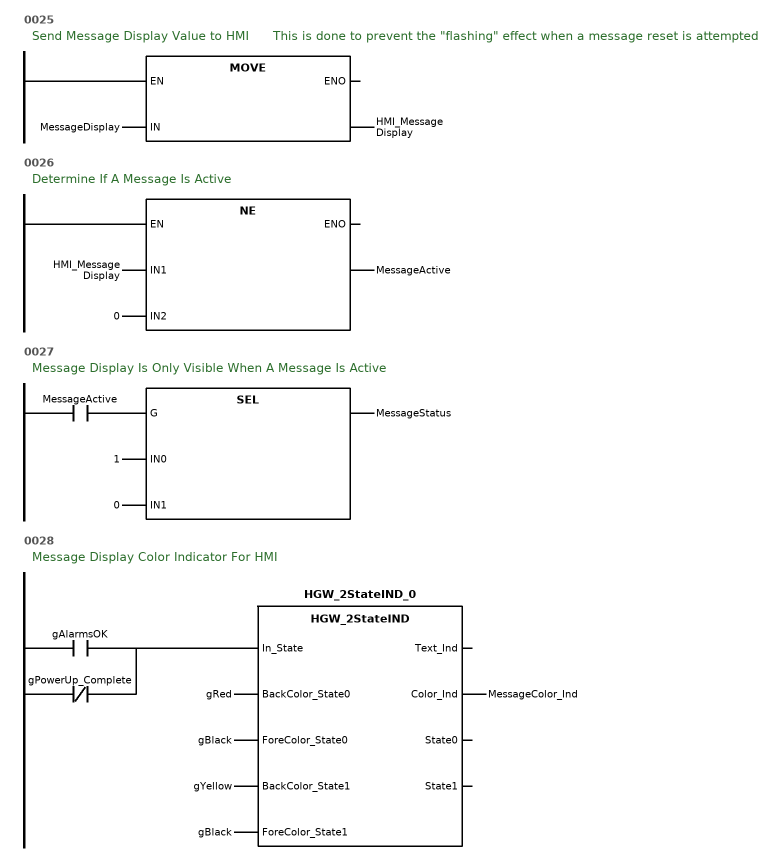
Ladder, written as Structured Text:
```iecst
(********************************************************************
 * COPYRIGHT --
 ********************************************************************
 * Program: Message_1
 * File: Message_1Cyclic.ld
 * Author: pkiel
 * Created: October 16, 2009
 ********************************************************************
 * Implementation of program Message_1
 ********************************************************************)

PROGRAM _CYCLIC
VAR
    _e1 : R_TRIG;
    _e2 : R_TRIG;
    _e3 : R_TRIG;
    _e4 : F_TRIG;
    _e5 : R_TRIG;
    _e6 : R_TRIG;
    _e7 : R_TRIG;
    _e8 : R_TRIG;
    _p9 : BOOL;
    _p10 : BOOL;
    _p11 : BOOL;
    _p12 : BOOL;
    _p13 : BOOL;
    _p14 : BOOL;
    _p15 : BOOL;
    _p16 : BOOL;
    _p17 : BOOL;
    _p18 : BOOL;
    _p19 : BOOL;
    _p20 : BOOL;
    _p21 : BOOL;
    _p22 : BOOL;
    _p23 : BOOL;
    _p24 : BOOL;
    _p25 : BOOL;
    _p26 : BOOL;
    _p27 : BOOL;
    _p28 : BOOL;
    _p29 : BOOL;
    _p30 : BOOL;
    _p31 : BOOL;
    _p32 : BOOL;
END_VAR
(* Network 1: Self Reset Timer *)
TON_0(IN := SelfReset, PT := t#3s);
IF TON_0.Q THEN SelfReset := FALSE; END_IF;

(* Network 2: Message Display Reset *)
_e1(CLK := gAlarmsOK);
_e2(CLK := gMachine_Run);
_e3(CLK := gHMI_Jog_PB);
_e4(CLK := SelfReset);
_e5(CLK := gQ_CR_MainPowerOn);
_e6(CLK := gAlarmReset);
_e7(CLK := g_bBundInit_OK);
_e8(CLK := gMachine_Jog);
MessageReset := _e1.Q OR _e2.Q OR _e3.Q OR _e4.Q OR _e5.Q OR _e6.Q OR _e7.Q OR _e8.Q;
IF _e1.Q OR _e2.Q OR _e3.Q OR _e4.Q OR _e5.Q OR _e6.Q OR _e7.Q OR _e8.Q THEN
    FirstMessage_L1 := FALSE;
    FirstMessage_L2 := FALSE;
    MessageDisplay := 0;
END_IF;

(* Network 3: ********** LEVEL 1 MESSAGES ********** (Used For Displaying Alarms)  Message #1: Machine Stop, E-Stop Alarm *)
_p9 := NOT gEStopAlarmsOK AND gQ_CR_MainPowerOn AND NOT FirstMessage_L1;
_p10 := Message[1] AND NOT MessageReset;
Message[1] := _p9 OR (Message[1] AND NOT MessageReset);
IF _p9 OR _p10 THEN
    FirstMessage_L1 := TRUE;
    MessageDisplay := 1;
END_IF;

(* Network 4: Message #2: Machine Stop, Guard Alarm *)
_p11 := NOT gGuardAlarmsOK AND gQ_CR_MainPowerOn AND NOT FirstMessage_L1;
_p12 := Message[2] AND NOT MessageReset;
Message[2] := _p11 OR (Message[2] AND NOT MessageReset);
IF _p11 OR _p12 THEN
    FirstMessage_L1 := TRUE;
    MessageDisplay := 2;
END_IF;

(* Network 5: Message #3: Machine Stop, Motor Alarm *)
_p13 := NOT gMotorAlarmsOK AND gQ_CR_MainPowerOn AND NOT FirstMessage_L1;
_p14 := Message[3] AND NOT MessageReset;
Message[3] := _p13 OR (Message[3] AND NOT MessageReset);
IF _p13 OR _p14 THEN
    FirstMessage_L1 := TRUE;
    MessageDisplay := 3;
END_IF;

(* Network 6: Message #4: Machine Stop, Jam Alarm *)
_p15 := NOT gJamAlarmsOK AND gQ_CR_MainPowerOn AND NOT FirstMessage_L1;
_p16 := Message[4] AND NOT MessageReset;
Message[4] := _p15 OR (Message[4] AND NOT MessageReset);
IF _p15 OR _p16 THEN
    FirstMessage_L1 := TRUE;
    MessageDisplay := 4;
END_IF;

(* Network 7: Message #5: Machine Stop, I/O Alarm *)
_p17 := NOT gIOAlarmsOK AND gQ_CR_MainPowerOn AND NOT FirstMessage_L1;
_p18 := Message[5] AND NOT MessageReset;
Message[5] := _p17 OR (Message[5] AND NOT MessageReset);
IF _p17 OR _p18 THEN
    FirstMessage_L1 := TRUE;
    MessageDisplay := 5;
END_IF;

(* Network 8: Message #6: Machine Stop, Web Break *)
_p19 := NOT gWebBreakAlarmsOK AND gQ_CR_MainPowerOn AND NOT FirstMessage_L1;
_p20 := Message[6] AND NOT MessageReset;
Message[6] := _p19 OR (Message[6] AND NOT MessageReset);
IF _p19 OR _p20 THEN
    FirstMessage_L1 := TRUE;
    MessageDisplay := 6;
END_IF;

(* Network 9: Message #30: Machine Stop, General alarm (230V Supply, Air, ...) *)
_p21 := NOT g_bGenAlarmsOK AND gQ_CR_MainPowerOn AND NOT FirstMessage_L1;
_p22 := Message[30] AND NOT MessageReset;
Message[30] := _p21 OR (Message[30] AND NOT MessageReset);
IF _p21 OR _p22 THEN
    FirstMessage_L1 := TRUE;
    MessageDisplay := 30;
END_IF;

(* Network 10: ********** LEVEL 2 MESSAGES ********** (Used For Displaying Machine Stops/Shutdowns)  Level 2 Permissives *)
Permissive_L2 := NOT FirstMessage_L1 AND gAlarmsOK;

(* Network 11: Message #21: Machine Stop, Unwind + Flexo Stop PB *)
_p23 := ((NOT gI_StopPB_1 AND NOT FirstMessage_L2) OR (Message[21] AND NOT MessageReset)) AND Permissive_L2;
Message[21] := _p23;
IF _p23 THEN
    FirstMessage_L2 := TRUE;
    MessageDisplay := 21;
END_IF;

(* Network 12: Message #22: Machine Stop, RS Stop PB *)
_p24 := ((NOT gI_StopPB_2 AND NOT FirstMessage_L2) OR (Message[22] AND NOT MessageReset)) AND Permissive_L2;
Message[22] := _p24;
IF _p24 THEN
    FirstMessage_L2 := TRUE;
    MessageDisplay := 22;
END_IF;

(* Network 13: Message #23: Machine Stop, Main Operator Station Stop PB *)
_p25 := ((NOT gI_StopPB_3 AND NOT FirstMessage_L2) OR (Message[23] AND NOT MessageReset)) AND Permissive_L2;
Message[23] := _p25;
IF _p25 THEN
    FirstMessage_L2 := TRUE;
    MessageDisplay := 23;
END_IF;

(* Network 14: Message #24: Machine Stop, Main Operator Station HMI Stop PB *)
_p26 := ((gHMI_Stop_PB AND NOT FirstMessage_L2) OR (Message[24] AND NOT MessageReset)) AND Permissive_L2;
Message[24] := _p26;
IF _p26 THEN
    FirstMessage_L2 := TRUE;
    MessageDisplay := 24;
END_IF;

(* Network 15: Message #25: Machine Stop, Unwind Low Roll Stop *)
_p27 := ((gUnwindLowRoll_Stop AND NOT FirstMessage_L2) OR (Message[25] AND NOT MessageReset)) AND Permissive_L2;
Message[25] := _p27;
IF _p27 THEN
    FirstMessage_L2 := TRUE;
    MessageDisplay := 25;
END_IF;

(* Network 16: Message #26: Machine Stop, Registration Missed Mark Shutdown *)
_p28 := ((gReg[5].ShutdownMissedMark AND NOT FirstMessage_L2) OR (Message[26] AND NOT MessageReset)) AND Permissive_L2;
Message[26] := _p28;
IF _p28 THEN
    FirstMessage_L2 := TRUE;
    MessageDisplay := 26;
END_IF;

(* Network 17: Message #27: Machine Stop, Registration Out Of Tolerance Shutdown *)
_p29 := ((gReg[5].ShutdownOutOfTolerance AND NOT FirstMessage_L2) OR (Message[27] AND NOT MessageReset)) AND Permissive_L2;
Message[27] := _p29;
IF _p29 THEN
    FirstMessage_L2 := TRUE;
    MessageDisplay := 27;
END_IF;

(* Network 18: Message #28: Machine Stop, Fast Stop PB *)
_p30 := ((NOT gI_FstopPB_1 AND NOT FirstMessage_L2) OR (Message[28] AND NOT MessageReset)) AND Permissive_L2;
Message[28] := _p30;
IF _p30 THEN
    FirstMessage_L2 := TRUE;
    MessageDisplay := 28;
END_IF;

(* Network 19: Message #29: Machine Stop, Bundler Stop PB *)
_p31 := ((NOT gI_Bund_Stop AND NOT FirstMessage_L2) OR (Message[29] AND NOT MessageReset)) AND Permissive_L2 AND g_bIndSelBundProd;
Message[29] := _p31;
IF _p31 THEN
    FirstMessage_L2 := TRUE;
    MessageDisplay := 29;
END_IF;

(* Network 20: ********** LEVEL 3 MESSAGES ********** (Used For Displaying General Warning Messages That Are Automatically Reset After 3 Seconds)  Level 3 Permissives *)
Permissive_L3 := NOT FirstMessage_L1 AND NOT FirstMessage_L2 AND gAlarmsOK;

(* Network 21: Message #51: Permissive Failure,  *)
_p32 := (((gHMI_Run_PB OR gI_PB_MachineStart) AND SparePermissive) OR (Message[51] AND NOT MessageReset)) AND Permissive_L3;
Message[51] := _p32;
IF _p32 THEN
    SelfReset := TRUE;
    MessageDisplay := 51;
END_IF;

(* Network 22: Message #98: System Drive Power Off *)
Message[98] := NOT g_bBundInit_OK;
IF NOT g_bBundInit_OK THEN MessageDisplay := 98; END_IF;

(* Network 23: Message #99: System Drive Power Off *)
Message[99] := gPowerUp_Complete AND NOT gQ_CR_MainPowerOn;
IF gPowerUp_Complete AND NOT gQ_CR_MainPowerOn THEN MessageDisplay := 99; END_IF;

(* Network 24: Message #100: Power Up Sequence Active *)
Message[100] := NOT gPowerUp_Complete;
IF NOT gPowerUp_Complete THEN MessageDisplay := 100; END_IF;

(* Network 25: Send Message Display Value to HMI      This is done to prevent the "flashing" effect when a message reset is attempted *)
HMI_MessageDisplay := MessageDisplay;

(* Network 26: Determine If A Message Is Active *)
MessageActive := HMI_MessageDisplay <> 0;

(* Network 27: Message Display Is Only Visible When A Message Is Active *)
MessageStatus := SEL(G := MessageActive, IN0 := 1, IN1 := 0);

(* Network 28: Message Display Color Indicator For HMI *)
HGW_2StateIND_0(In_State := gAlarmsOK OR NOT gPowerUp_Complete, BackColor_State0 := gRed, ForeColor_State0 := gBlack, BackColor_State1 := gYellow, ForeColor_State1 := gBlack);
MessageColor_Ind := HGW_2StateIND_0.Color_Ind;
END_PROGRAM
```

### Program Logical/HMI/Message_2 (IEC) - Message Display #2 Code

#### Message_2.var
```iecst
(********************************************************************
 * COPYRIGHT --
 ********************************************************************
 * Program: Message_2
 * File: Message_2.var
 * Author: pkiel
 * Created: October 26, 2009
 ********************************************************************
 * Local variables of program Message_2
 ********************************************************************)
VAR
	AxisReadyPermissive : BOOL;
	FirstMessage : BOOL;
	FirstMessage_L1 : BOOL;
	FirstMessage_L2 : BOOL;
	HGW_Toggle_0 : HGW_Toggle;
	HMI_MessageDisplay : INT;
	Message : ARRAY[0..100] OF BOOL;
	MessageActive : BOOL;
	MessageDisplay : UINT;
	MessageReset : BOOL;
	MessageStatus : UINT;
	Permissive_L2 : BOOL;
	Permissive_L3 : BOOL;
	SelfReset : BOOL;
	TON_0 : TON;
END_VAR
```

#### Message_2Cyclic.ld
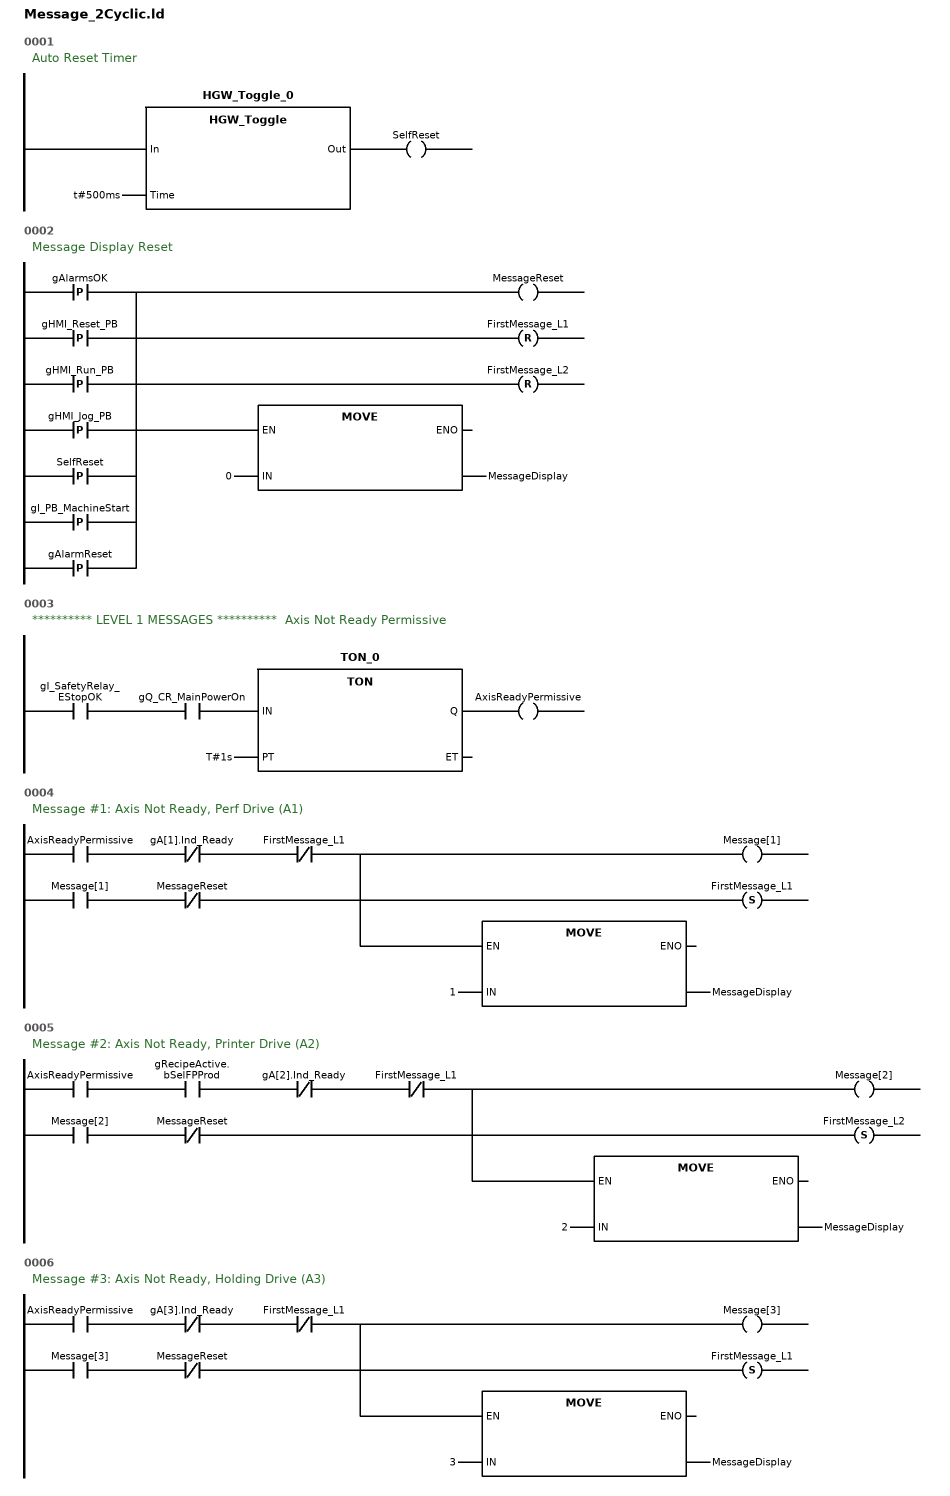
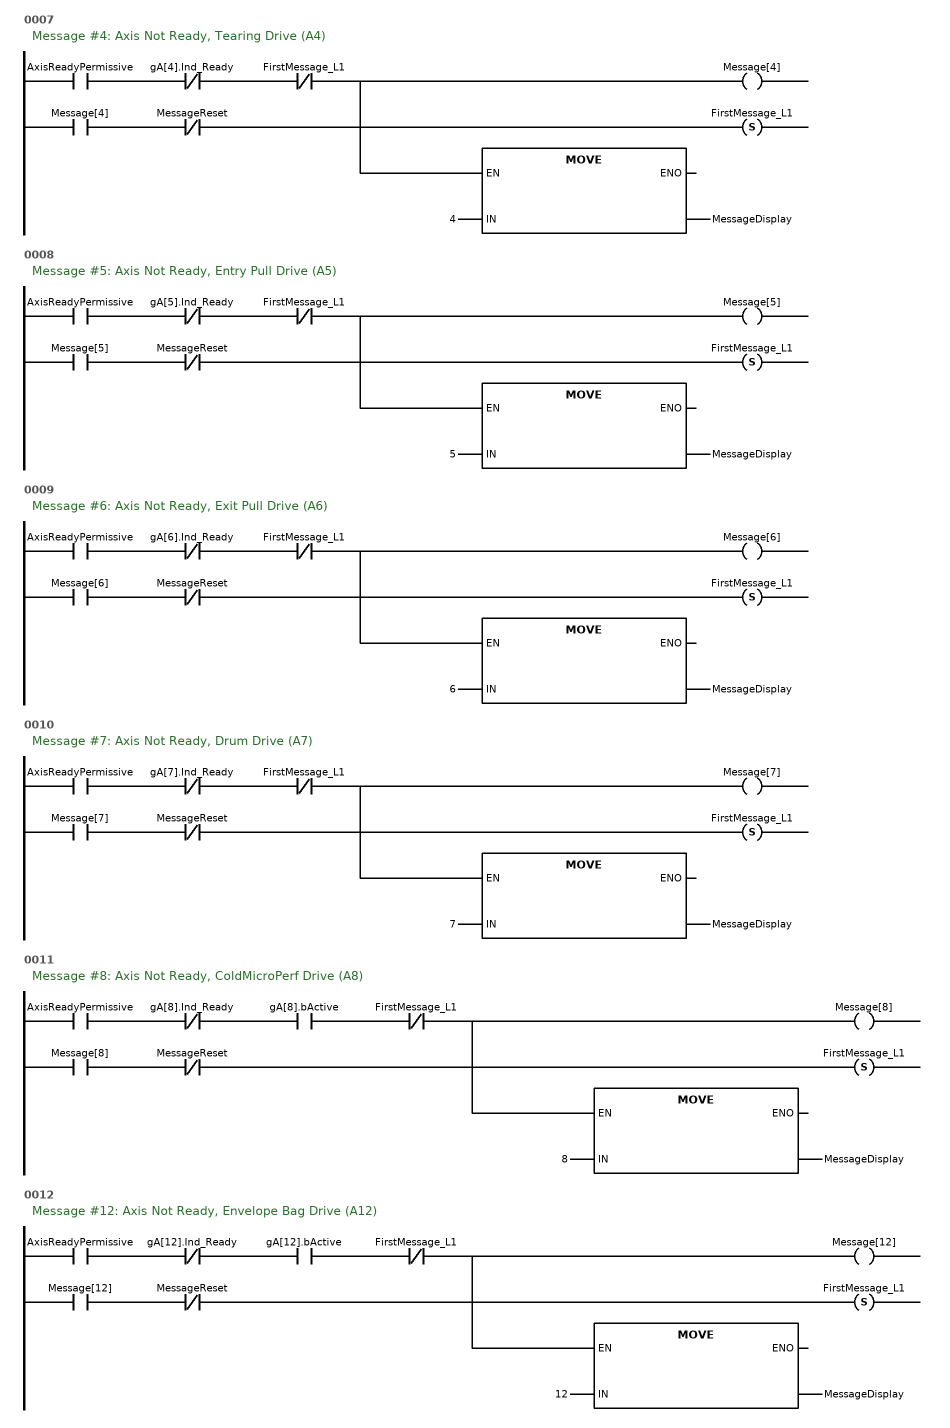
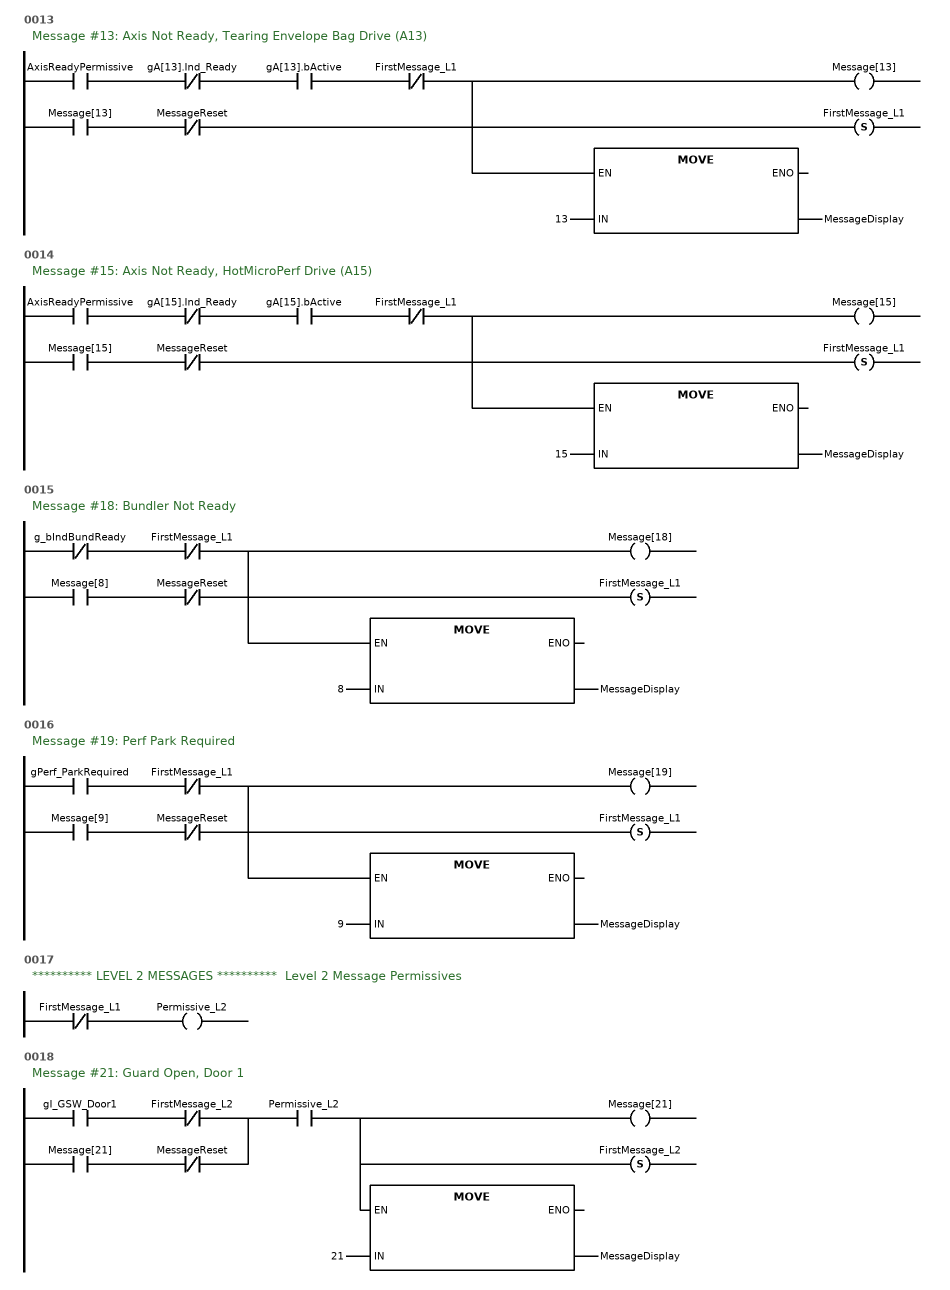
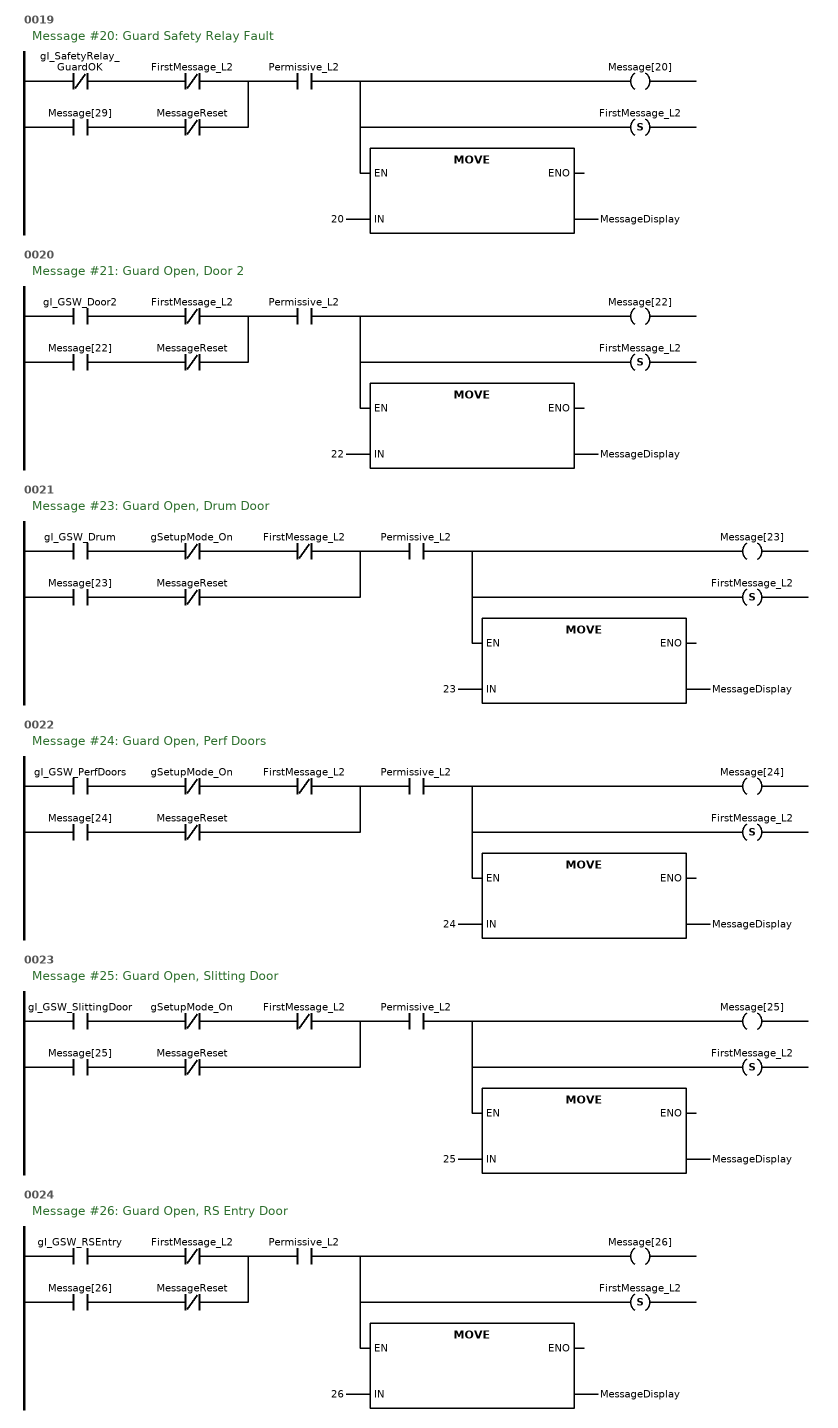
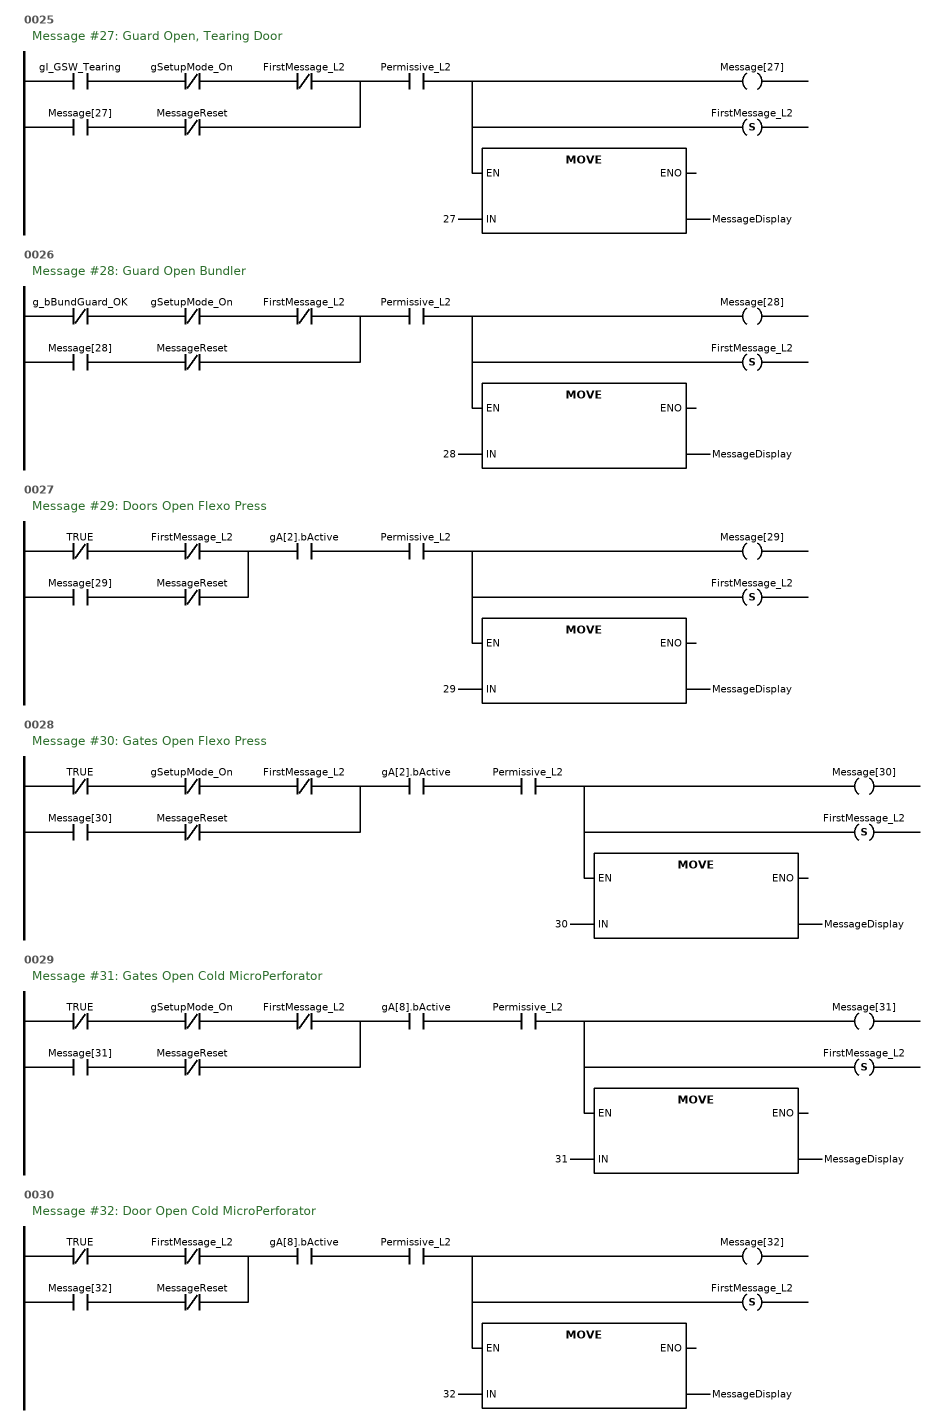
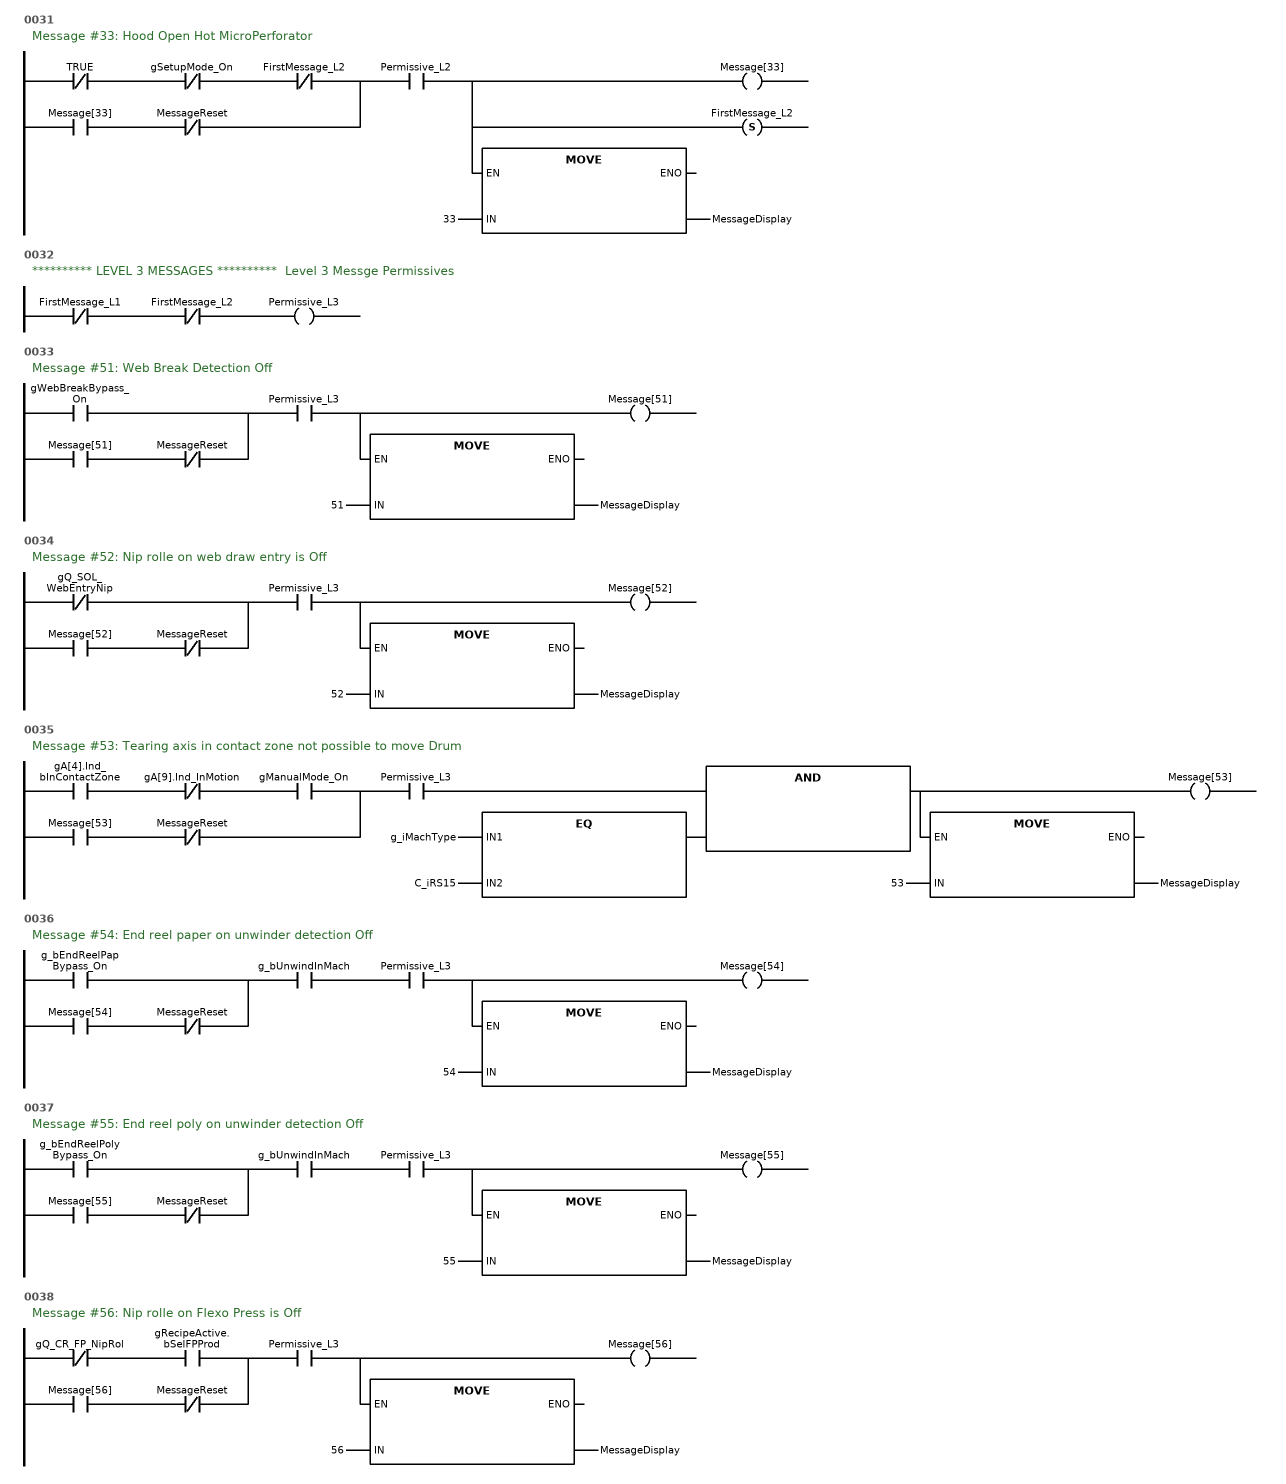
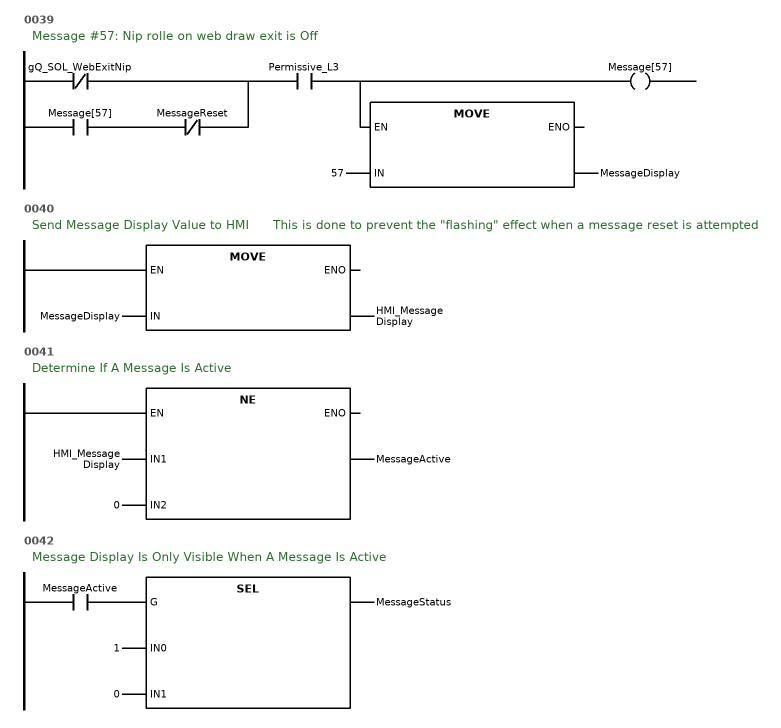
Ladder, written as Structured Text:
```iecst
(********************************************************************
 * COPYRIGHT --
 ********************************************************************
 * Program: Message_2
 * File: Message_2Cyclic.ld
 * Author: pkiel
 * Created: October 26, 2009
 ********************************************************************
 * Implementation of program Message_2
 ********************************************************************)

PROGRAM _CYCLIC
VAR
    _e1 : R_TRIG;
    _e2 : R_TRIG;
    _e3 : R_TRIG;
    _e4 : R_TRIG;
    _e5 : R_TRIG;
    _e6 : R_TRIG;
    _e7 : R_TRIG;
    _p8 : BOOL;
    _p9 : BOOL;
    _p10 : BOOL;
    _p11 : BOOL;
    _p12 : BOOL;
    _p13 : BOOL;
    _p14 : BOOL;
    _p15 : BOOL;
    _p16 : BOOL;
    _p17 : BOOL;
    _p18 : BOOL;
    _p19 : BOOL;
    _p20 : BOOL;
    _p21 : BOOL;
    _p22 : BOOL;
    _p23 : BOOL;
    _p24 : BOOL;
    _p25 : BOOL;
    _p26 : BOOL;
    _p27 : BOOL;
    _p28 : BOOL;
    _p29 : BOOL;
    _p30 : BOOL;
    _p31 : BOOL;
    _p32 : BOOL;
    _p33 : BOOL;
    _p34 : BOOL;
    _p35 : BOOL;
    _p36 : BOOL;
    _p37 : BOOL;
    _p38 : BOOL;
    _p39 : BOOL;
    _p40 : BOOL;
    _p41 : BOOL;
    _p42 : BOOL;
    _p43 : BOOL;
    _p44 : BOOL;
    _p45 : BOOL;
    _p46 : BOOL;
    _p47 : BOOL;
    _p48 : BOOL;
    _p49 : BOOL;
    _t50 : BOOL;
    _p51 : BOOL;
    _p52 : BOOL;
    _p53 : BOOL;
    _p54 : BOOL;
END_VAR
(* Network 1: Auto Reset Timer *)
HGW_Toggle_0(In := TRUE, Time := t#500ms);
SelfReset := HGW_Toggle_0.Out;

(* Network 2: Message Display Reset *)
_e1(CLK := gAlarmsOK);
_e2(CLK := gHMI_Reset_PB);
_e3(CLK := gHMI_Run_PB);
_e4(CLK := gHMI_Jog_PB);
_e5(CLK := SelfReset);
_e6(CLK := gI_PB_MachineStart);
_e7(CLK := gAlarmReset);
MessageReset := _e1.Q OR _e2.Q OR _e3.Q OR _e4.Q OR _e5.Q OR _e6.Q OR _e7.Q;
IF _e1.Q OR _e2.Q OR _e3.Q OR _e4.Q OR _e5.Q OR _e6.Q OR _e7.Q THEN
    FirstMessage_L1 := FALSE;
    FirstMessage_L2 := FALSE;
    MessageDisplay := 0;
END_IF;

(* Network 3: ********** LEVEL 1 MESSAGES **********  Axis Not Ready Permissive *)
TON_0(IN := gI_SafetyRelay_EStopOK AND gQ_CR_MainPowerOn, PT := T#1s);
AxisReadyPermissive := TON_0.Q;

(* Network 4: Message #1: Axis Not Ready, Perf Drive (A1) *)
_p8 := AxisReadyPermissive AND NOT gA[1].Ind_Ready AND NOT FirstMessage_L1;
_p9 := Message[1] AND NOT MessageReset;
Message[1] := _p8 OR (Message[1] AND NOT MessageReset);
IF _p8 OR _p9 THEN
    FirstMessage_L1 := TRUE;
    MessageDisplay := 1;
END_IF;

(* Network 5: Message #2: Axis Not Ready, Printer Drive (A2) *)
_p10 := AxisReadyPermissive AND gRecipeActive.bSelFPProd AND NOT gA[2].Ind_Ready AND NOT FirstMessage_L1;
_p11 := Message[2] AND NOT MessageReset;
Message[2] := _p10 OR (Message[2] AND NOT MessageReset);
IF _p10 OR _p11 THEN
    FirstMessage_L2 := TRUE;
    MessageDisplay := 2;
END_IF;

(* Network 6: Message #3: Axis Not Ready, Holding Drive (A3) *)
_p12 := AxisReadyPermissive AND NOT gA[3].Ind_Ready AND NOT FirstMessage_L1;
_p13 := Message[3] AND NOT MessageReset;
Message[3] := _p12 OR (Message[3] AND NOT MessageReset);
IF _p12 OR _p13 THEN
    FirstMessage_L1 := TRUE;
    MessageDisplay := 3;
END_IF;

(* Network 7: Message #4: Axis Not Ready, Tearing Drive (A4) *)
_p14 := AxisReadyPermissive AND NOT gA[4].Ind_Ready AND NOT FirstMessage_L1;
_p15 := Message[4] AND NOT MessageReset;
Message[4] := _p14 OR (Message[4] AND NOT MessageReset);
IF _p14 OR _p15 THEN
    FirstMessage_L1 := TRUE;
    MessageDisplay := 4;
END_IF;

(* Network 8: Message #5: Axis Not Ready, Entry Pull Drive (A5) *)
_p16 := AxisReadyPermissive AND NOT gA[5].Ind_Ready AND NOT FirstMessage_L1;
_p17 := Message[5] AND NOT MessageReset;
Message[5] := _p16 OR (Message[5] AND NOT MessageReset);
IF _p16 OR _p17 THEN
    FirstMessage_L1 := TRUE;
    MessageDisplay := 5;
END_IF;

(* Network 9: Message #6: Axis Not Ready, Exit Pull Drive (A6) *)
_p18 := AxisReadyPermissive AND NOT gA[6].Ind_Ready AND NOT FirstMessage_L1;
_p19 := Message[6] AND NOT MessageReset;
Message[6] := _p18 OR (Message[6] AND NOT MessageReset);
IF _p18 OR _p19 THEN
    FirstMessage_L1 := TRUE;
    MessageDisplay := 6;
END_IF;

(* Network 10: Message #7: Axis Not Ready, Drum Drive (A7) *)
_p20 := AxisReadyPermissive AND NOT gA[7].Ind_Ready AND NOT FirstMessage_L1;
_p21 := Message[7] AND NOT MessageReset;
Message[7] := _p20 OR (Message[7] AND NOT MessageReset);
IF _p20 OR _p21 THEN
    FirstMessage_L1 := TRUE;
    MessageDisplay := 7;
END_IF;

(* Network 11: Message #8: Axis Not Ready, ColdMicroPerf Drive (A8) *)
_p22 := AxisReadyPermissive AND NOT gA[8].Ind_Ready AND gA[8].bActive AND NOT FirstMessage_L1;
_p23 := Message[8] AND NOT MessageReset;
Message[8] := _p22 OR (Message[8] AND NOT MessageReset);
IF _p22 OR _p23 THEN
    FirstMessage_L1 := TRUE;
    MessageDisplay := 8;
END_IF;

(* Network 12: Message #12: Axis Not Ready, Envelope Bag Drive (A12) *)
_p24 := AxisReadyPermissive AND NOT gA[12].Ind_Ready AND gA[12].bActive AND NOT FirstMessage_L1;
_p25 := Message[12] AND NOT MessageReset;
Message[12] := _p24 OR (Message[12] AND NOT MessageReset);
IF _p24 OR _p25 THEN
    FirstMessage_L1 := TRUE;
    MessageDisplay := 12;
END_IF;

(* Network 13: Message #13: Axis Not Ready, Tearing Envelope Bag Drive (A13) *)
_p26 := AxisReadyPermissive AND NOT gA[13].Ind_Ready AND gA[13].bActive AND NOT FirstMessage_L1;
_p27 := Message[13] AND NOT MessageReset;
Message[13] := _p26 OR (Message[13] AND NOT MessageReset);
IF _p26 OR _p27 THEN
    FirstMessage_L1 := TRUE;
    MessageDisplay := 13;
END_IF;

(* Network 14: Message #15: Axis Not Ready, HotMicroPerf Drive (A15) *)
_p28 := AxisReadyPermissive AND NOT gA[15].Ind_Ready AND gA[15].bActive AND NOT FirstMessage_L1;
_p29 := Message[15] AND NOT MessageReset;
Message[15] := _p28 OR (Message[15] AND NOT MessageReset);
IF _p28 OR _p29 THEN
    FirstMessage_L1 := TRUE;
    MessageDisplay := 15;
END_IF;

(* Network 15: Message #18: Bundler Not Ready *)
_p30 := Message[8] AND NOT MessageReset;
Message[18] := (NOT g_bIndBundReady AND NOT FirstMessage_L1) OR (Message[8] AND NOT MessageReset);
_p31 := NOT g_bIndBundReady AND NOT FirstMessage_L1;
IF (NOT g_bIndBundReady AND NOT FirstMessage_L1) OR _p30 THEN FirstMessage_L1 := TRUE; END_IF;
IF _p31 OR _p30 THEN MessageDisplay := 8; END_IF;

(* Network 16: Message #19: Perf Park Required *)
_p32 := Message[9] AND NOT MessageReset;
Message[19] := (gPerf_ParkRequired AND NOT FirstMessage_L1) OR (Message[9] AND NOT MessageReset);
_p33 := gPerf_ParkRequired AND NOT FirstMessage_L1;
IF (gPerf_ParkRequired AND NOT FirstMessage_L1) OR _p32 THEN FirstMessage_L1 := TRUE; END_IF;
IF _p33 OR _p32 THEN MessageDisplay := 9; END_IF;

(* Network 17: ********** LEVEL 2 MESSAGES **********  Level 2 Message Permissives *)
Permissive_L2 := NOT FirstMessage_L1;

(* Network 18: Message #21: Guard Open, Door 1 *)
_p34 := ((gI_GSW_Door1 AND NOT FirstMessage_L2) OR (Message[21] AND NOT MessageReset)) AND Permissive_L2;
Message[21] := _p34;
IF _p34 THEN
    FirstMessage_L2 := TRUE;
    MessageDisplay := 21;
END_IF;

(* Network 19: Message #20: Guard Safety Relay Fault *)
_p35 := ((NOT gI_SafetyRelay_GuardOK AND NOT FirstMessage_L2) OR (Message[29] AND NOT MessageReset)) AND Permissive_L2;
Message[20] := _p35;
IF _p35 THEN
    FirstMessage_L2 := TRUE;
    MessageDisplay := 20;
END_IF;

(* Network 20: Message #21: Guard Open, Door 2 *)
_p36 := ((gI_GSW_Door2 AND NOT FirstMessage_L2) OR (Message[22] AND NOT MessageReset)) AND Permissive_L2;
Message[22] := _p36;
IF _p36 THEN
    FirstMessage_L2 := TRUE;
    MessageDisplay := 22;
END_IF;

(* Network 21: Message #23: Guard Open, Drum Door *)
_p37 := ((gI_GSW_Drum AND NOT gSetupMode_On AND NOT FirstMessage_L2) OR (Message[23] AND NOT MessageReset)) AND Permissive_L2;
Message[23] := _p37;
IF _p37 THEN
    FirstMessage_L2 := TRUE;
    MessageDisplay := 23;
END_IF;

(* Network 22: Message #24: Guard Open, Perf Doors *)
_p38 := ((gI_GSW_PerfDoors AND NOT gSetupMode_On AND NOT FirstMessage_L2) OR (Message[24] AND NOT MessageReset)) AND Permissive_L2;
Message[24] := _p38;
IF _p38 THEN
    FirstMessage_L2 := TRUE;
    MessageDisplay := 24;
END_IF;

(* Network 23: Message #25: Guard Open, Slitting Door *)
_p39 := ((gI_GSW_SlittingDoor AND NOT gSetupMode_On AND NOT FirstMessage_L2) OR (Message[25] AND NOT MessageReset)) AND Permissive_L2;
Message[25] := _p39;
IF _p39 THEN
    FirstMessage_L2 := TRUE;
    MessageDisplay := 25;
END_IF;

(* Network 24: Message #26: Guard Open, RS Entry Door *)
_p40 := ((gI_GSW_RSEntry AND NOT FirstMessage_L2) OR (Message[26] AND NOT MessageReset)) AND Permissive_L2;
Message[26] := _p40;
IF _p40 THEN
    FirstMessage_L2 := TRUE;
    MessageDisplay := 26;
END_IF;

(* Network 25: Message #27: Guard Open, Tearing Door *)
_p41 := ((gI_GSW_Tearing AND NOT gSetupMode_On AND NOT FirstMessage_L2) OR (Message[27] AND NOT MessageReset)) AND Permissive_L2;
Message[27] := _p41;
IF _p41 THEN
    FirstMessage_L2 := TRUE;
    MessageDisplay := 27;
END_IF;

(* Network 26: Message #28: Guard Open Bundler *)
_p42 := ((NOT g_bBundGuard_OK AND NOT gSetupMode_On AND NOT FirstMessage_L2) OR (Message[28] AND NOT MessageReset)) AND Permissive_L2;
Message[28] := _p42;
IF _p42 THEN
    FirstMessage_L2 := TRUE;
    MessageDisplay := 28;
END_IF;

(* Network 27: Message #29: Doors Open Flexo Press *)
_p43 := Message[29] AND NOT MessageReset AND gA[2].bActive AND Permissive_L2;
Message[29] := _p43;
IF _p43 THEN
    FirstMessage_L2 := TRUE;
    MessageDisplay := 29;
END_IF;

(* Network 28: Message #30: Gates Open Flexo Press *)
_p44 := Message[30] AND NOT MessageReset AND gA[2].bActive AND Permissive_L2;
Message[30] := _p44;
IF _p44 THEN
    FirstMessage_L2 := TRUE;
    MessageDisplay := 30;
END_IF;

(* Network 29: Message #31: Gates Open Cold MicroPerforator  *)
_p45 := Message[31] AND NOT MessageReset AND gA[8].bActive AND Permissive_L2;
Message[31] := _p45;
IF _p45 THEN
    FirstMessage_L2 := TRUE;
    MessageDisplay := 31;
END_IF;

(* Network 30: Message #32: Door Open Cold MicroPerforator  *)
_p46 := Message[32] AND NOT MessageReset AND gA[8].bActive AND Permissive_L2;
Message[32] := _p46;
IF _p46 THEN
    FirstMessage_L2 := TRUE;
    MessageDisplay := 32;
END_IF;

(* Network 31: Message #33: Hood Open Hot MicroPerforator  *)
_p47 := Message[33] AND NOT MessageReset AND Permissive_L2;
Message[33] := _p47;
IF _p47 THEN
    FirstMessage_L2 := TRUE;
    MessageDisplay := 33;
END_IF;

(* Network 32: ********** LEVEL 3 MESSAGES **********  Level 3 Messge Permissives *)
Permissive_L3 := NOT FirstMessage_L1 AND NOT FirstMessage_L2;

(* Network 33: Message #51: Web Break Detection Off *)
_p48 := (gWebBreakBypass_On OR (Message[51] AND NOT MessageReset)) AND Permissive_L3;
Message[51] := _p48;
IF _p48 THEN MessageDisplay := 51; END_IF;

(* Network 34: Message #52: Nip rolle on web draw entry is Off  *)
_p49 := (NOT gQ_SOL_WebEntryNip OR (Message[52] AND NOT MessageReset)) AND Permissive_L3;
Message[52] := _p49;
IF _p49 THEN MessageDisplay := 52; END_IF;

(* Network 35: Message #53: Tearing axis in contact zone not possible to move Drum *)
_t50 := (((gA[4].Ind_bInContactZone AND NOT gA[9].Ind_InMotion AND gManualMode_On) OR (Message[53] AND NOT MessageReset)) AND Permissive_L3) AND (g_iMachType = C_iRS15);
Message[53] := _t50;
IF _t50 THEN MessageDisplay := 53; END_IF;

(* Network 36: Message #54: End reel paper on unwinder detection Off *)
_p51 := (g_bEndReelPapBypass_On OR (Message[54] AND NOT MessageReset)) AND g_bUnwindInMach AND Permissive_L3;
Message[54] := _p51;
IF _p51 THEN MessageDisplay := 54; END_IF;

(* Network 37: Message #55: End reel poly on unwinder detection Off *)
_p52 := (g_bEndReelPolyBypass_On OR (Message[55] AND NOT MessageReset)) AND g_bUnwindInMach AND Permissive_L3;
Message[55] := _p52;
IF _p52 THEN MessageDisplay := 55; END_IF;

(* Network 38: Message #56: Nip rolle on Flexo Press is Off *)
_p53 := ((NOT gQ_CR_FP_NipRol AND gRecipeActive.bSelFPProd) OR (Message[56] AND NOT MessageReset)) AND Permissive_L3;
Message[56] := _p53;
IF _p53 THEN MessageDisplay := 56; END_IF;

(* Network 39: Message #57: Nip rolle on web draw exit is Off  *)
_p54 := (NOT gQ_SOL_WebExitNip OR (Message[57] AND NOT MessageReset)) AND Permissive_L3;
Message[57] := _p54;
IF _p54 THEN MessageDisplay := 57; END_IF;

(* Network 40: Send Message Display Value to HMI      This is done to prevent the "flashing" effect when a message reset is attempted *)
HMI_MessageDisplay := MessageDisplay;

(* Network 41: Determine If A Message Is Active *)
MessageActive := HMI_MessageDisplay <> 0;

(* Network 42: Message Display Is Only Visible When A Message Is Active *)
MessageStatus := SEL(G := MessageActive, IN0 := 1, IN1 := 0);
END_PROGRAM
```

### Program Logical/HMI/BackUp (IEC) - Variable Back Up Routine

#### BackUpInit.st
```iecst
(********************************************************************
 * COPYRIGHT --
 ********************************************************************
 * Program: BackUp
 * File: BackUpInit.st
 * Author: pkiel
 * Created: December 11, 2009
 ********************************************************************
 * Implementation of program BackUp
 ********************************************************************)

PROGRAM _INIT

strDevice       := 'USB1';
strFile         := 'SystemBackup.dat';
byStep			:= 0;
bOK				:= 1;

END_PROGRAM
```

### Program Logical/HMI/CPURestart (IEC) - A new program

#### CPURestart.var - Local variables
```iecst
(********************************************************************
 * COPYRIGHT -- .
 ********************************************************************
 * Program: CPURestart
 * File: CPURestart.var
 * Author: dominique
 * Created: March 18, 2012
 ********************************************************************
 * Local variables of program CPURestart
 ********************************************************************)

VAR RETAIN

  HMI_iCRestartStat : INT ;
  HMI_iWRestartStat : INT ;

END_VAR

VAR

  HMI_CmdColdRestart : BOOL ;
  uiRetColdRestart   : UINT ;
  HMI_CmdWarmRestart : BOOL ;
  uiRetWarmRestart   : UINT ;

END_VAR

VAR CONSTANT

END_VAR
```

- Visualisation Logical/HMI/HMI_10 (not shown)

### Program Logical/BagMachine_Section/MasterAxis/A9_Init/A9_Basic

#### A9_BasicInit.st
```iecst
(********************************************************************
 * COPYRIGHT -- Microsoft
 ********************************************************************
 * Program: A9_Basic
 * File: A9_BasicInit.st
 * Author: pkiel
 * Created: July 12, 2011
 ********************************************************************
 * Implementation of program A9_Basic
 ********************************************************************)

PROGRAM _INIT

	(* Axis Setpoint Variables *)
		gA[9].SP_MotorPPR := 36000;
		gA[9].SP_GearBoxInput:= 1;
		gA[9].SP_GearBoxOutput:= 1;
		gA[9].AxisPeriod := (gA[9].SP_MotorPPR*gA[9].SP_GearBoxInput/gA[9].SP_GearBoxOutput);
		gA[9].UnitsPerDeg := gA[9].AxisPeriod/360;
		gA[9].SP_Decel := 0.4*gA[9].AxisPeriod;
		gA[9].SP_EStopDecel := 3.0*gA[9].AxisPeriod;
		gA[9].SP_FStopDecel := 1.5*gA[9].AxisPeriod;
		gA[9].SP_GenFaultDecel := 1.5*gA[9].AxisPeriod;
		gA[9].SP_GuardFaultDecel := 1.5*gA[9].AxisPeriod;
		gA[9].SP_WebBreakDecel := 1.5*gA[9].AxisPeriod;
		gA[9].HomeVelocity:=12*gA[9].AxisPeriod/60.0;

	(* access master axis *)
		AxisErrorNcAccess := ncaccess(ncACP10MAN, ADR('Axis9'), ADR(gA[9].Ident));

	(* Trigger Initialization Of ModPosition *)
		InitModPosition:=1;

END_PROGRAM
```

- Data object Logical/BagMachine_Section/MasterAxis/A9_Init/A9_Init (Vax) (no source held here)

- Data object Logical/BagMachine_Section/MasterAxis/A9_Init/A9_Par (Apt) (no source held here)

### Program Logical/BagMachine_Section/MasterAxis/A9_Init/SetSpeedMode

#### SetSpeedModeCyclic.st
```iecst
(********************************************************************
 * COPYRIGHT -- .
 ********************************************************************
 * Program: SetSpeedMode
 * File: SetSpeedModeCyclic.st
 * Author: dominique
 * Created: September 29, 2011
 ********************************************************************
 * Implementation of program SetSpeedMode
 ********************************************************************)

PROGRAM _CYCLIC

// Select set speed mode
  IF HMI_bSetSpeed_PB THEN
    IF NOT(gr_bSetSpeedMode) THEN
      gr_bSetSpeedMode := 1 ; // Set MANU
    ELSE
      HMI_uiConfirmSetSpeedVisibl := 0 ; // Display PopUp confirm set AUTO
    END_IF ;
    HMI_bSetSpeed_PB := 0 ;
  END_IF ;

END_PROGRAM
```

#### SetSpeedModeInit.st
```iecst
(********************************************************************
 * COPYRIGHT -- .
 ********************************************************************
 * Program: SetSpeedMode
 * File: SetSpeedModeInit.st
 * Author: dominique
 * Created: September 29, 2011
 ********************************************************************
 * Implementation of program SetSpeedMode
 ********************************************************************)

PROGRAM _INIT
  HMI_uiConfirmSetSpeedVisibl := 1 ;
END_PROGRAM
```

### Package Logical/BagMachine_Section/Servo_Power_Supply/Axis0 - Servo Power Supply

### Program Logical/BagMachine_Section/Servo_Power_Supply/Axis0/A0_Basic (IEC)

#### A0_BasicInit.st - Initialization code
```iecst
(********************************************************************
 * COPYRIGHT -- Microsoft
 ********************************************************************
 * Program: A0_Basic
 * File: A0_BasicInit.st
 * Author: pkiel
 * Created: July 17, 2011
 ********************************************************************
 * Implementation of program A0_Basic
 ********************************************************************)

PROGRAM _INIT

	(* access master axis *)
		AxisErrorNcAccess := ncaccess(ncACP10MAN, ADR('Axis0'), ADR(gA[0].Ident));

END_PROGRAM
```

#### A0_Basic.var - Local variables
```iecst
(********************************************************************
 * COPYRIGHT -- Microsoft
 ********************************************************************
 * Program: A0_Basic
 * File: A0_Basic.var
 * Author: pkiel
 * Created: July 17, 2011
 ********************************************************************
 * Local variables of program A0_Basic
 ********************************************************************)
VAR
	AutoAck : BOOL;
	AxisErrorNcAccess : UINT;
	DriveStatus : MC_DRIVESTATUS_TYP;
	MC_BR_PowerMeter_0 : MC_BR_PowerMeter;
	MC_BR_ReadDriveStatus_0 : MC_BR_ReadDriveStatus;
	MC_Power_0 : MC_Power;
	MC_ReadAxisError_0 : MC_ReadAxisError;
	MC_ReadStatus_0 : MC_ReadStatus;
	MC_Reset_0 : MC_Reset;
  rRepeatMetric : REAL ;
END_VAR
```

### A0_Par.apt
```
AcoposParameterTable:
  Root Parameters:
    110 = ncSW_OFF (Name=CMD_SIMULATION)  // Simulation mode: Command
    128 = 1 (Name=SGEN_SW_END_IGNORE)  // Limit values: Ignore SW end positions
    10 = 50 (Name=R_BLEEDER_EXT, Unit=Ohm)  // Bleeder: External: Resistance
    11 = 682.85 (Name=TEMP_MAX_BLEEDER_EXT, Unit=°C)  // Bleeder: External: Limit temperature
    12 = 1.517 (Name=RTH_BLEEDER_AMB_EXT, Unit=°C/W)  // Bleeder: External: Thermic resistance
    13 = 16.3 (Name=CTH_BLEEDER_EXT, Unit=Ws/°C)  // Bleeder: External: Thermic capacity
    398 = 1 (Name=BLEEDER_SELECTOR_EXT)  // Bleeder: Selector
```

### Package Logical/BagMachine_Section/Perf - Axis

### Program Logical/BagMachine_Section/Perf/Axis1/A1_Automat (IEC)

#### A1_AutomatCyclic.st - Cyclic code
```iecst
(********************************************************************
 * COPYRIGHT -- Microsoft
 ********************************************************************
 * Program: A1_Automat
 * File: A1_AutomatCyclic.st
 * Author: pkiel
 * Created: July 12, 2011
 ********************************************************************
 * Implementation of program A1_Automat
 ********************************************************************)

PROGRAM _CYCLIC

  // Synchro ratio Master/Slave
     // Master = Virtuel Perf
     gA[1].rRSynNum := 1 ;
     gA[1].rRSynDen := 1 ;

(**** PROFILED CAM AUTOMAT WITH ABSOLUTE PHASE SYNCHRONIZATION FOR PERF AXIS ***)

(* Set Up Master Position Parameter ID *)
	Synch_Request := gA[1].Cmd_SynchronizedMotion;
	IF (Synch_Request AND NOT ParID_Ready) THEN
		  MC_BR_InitMasterParIDTransfer_0.Master:=gA[11].Ident;
	    MC_BR_InitMasterParIDTransfer_0.Slave:=gA[1].Ident;
	    MC_BR_InitMasterParIDTransfer_0.MasterParID:=412;   // 412: VAX: Position, S_SET_VAX1, DINT
	    MC_BR_InitMasterParIDTransfer_0.SlaveChannel:=1;
	    MC_BR_InitMasterParIDTransfer_0.Execute:=TRUE;
	    IF (MC_BR_InitMasterParIDTransfer_0.Done) THEN
	      MasterParID:=MC_BR_InitMasterParIDTransfer_0.ReceiveParID;
	      MC_BR_InitMasterParIDTransfer_0.Execute:=FALSE;
	      ParID_Ready:=1;
	    ELSIF (MC_BR_InitMasterParIDTransfer_0.Error) THEN
	    (*Store ErrorID in a variable,
	      ErrorID is reset on falling edge of 'Execute'*)
	      ErrorID:=MC_BR_InitMasterParIDTransfer_0.ErrorID;
	      ParID_Ready:=0;
	      MC_BR_InitMasterParIDTransfer_0.Execute:=FALSE;
	    END_IF
	END_IF
	MC_BR_InitMasterParIDTransfer_0();

(**** Initialize Automat Parameters Upon Automat Start Request ****)
  bInitCamAuto := ParID_Ready    AND
                  g_bCameProf_OK AND
                  1              ;

	IF (EDGEPOS(bInitCamAuto))THEN

		//general automat parameter
			//AutData.Master		    := gA[1].Ident;
			AutData.MasterParID		  := MasterParID;
			AutData.StartPosition		:= 0;
			AutData.StartInterval		:= gA[11].AxisPeriod;
			AutData.MaxMasterVelocity	:= gr_rMachMaxSpeed_BPM ;

		//**** Calculations ***
      IF gRecipeActive.bSelEnvBProd THEN
        //MatchedSpeed_Inch := gSP_A[1].MatchedSpeed/360.0*g_rActualSizePerf_in ;  // D.M. Le 10/01/2012 Pyrollpack_14661   Replaced by the line below because operator is able to change the size of the Perf => the length of matched speed is constant
        MatchedSpeed_Inch := gSP_EnvBPerf.rZoneBefPerf_in + gSP_EnvBPerf.rZoneAftPerf_in ;
      ELSE
        //MatchedSpeed_Inch := gSP_A[1].MatchedSpeed/360.0*g_rActualSizePerf_in ;  // D.M. Le 10/01/2012 Pyrollpack_14661   Replaced by the line below because operator is able to change the size of the Perf => the length of matched speed is constant
        MatchedSpeed_Inch := gSP_StandPerf.rZoneBefPerf_in + gSP_StandPerf.rZoneAftPerf_in ;
      END_IF
			MasterOffset      := 0 ;
			Slave_AxisPeriod  := gA[1].AxisPeriod/gSP_PerfKnifeCount ;

		//**** Slave Starting In Matched Speed Zone ***
      IF g_bPerfInMatchedSpeed THEN
        InMatched := 1;

			//Automat STATE 0 Basis State
        AutData.State[0].Event[0].Type      := ncST_END;
        AutData.State[0].Event[0].Attribute := ncAT_ONCE;
        AutData.State[0].Event[0].NextState := 1;

        rTempPosA1_Inch := H_FC_Modulus(IN_rMod:=360*gA[1].InchPerDeg/gSP_PerfKnifeCount, IN_rVar:=gA[1].PositionInch) ;

			//Initial Matched Speed Zone
				AutData.State[1].CamProfileIndex := 16#FFFF;
				AutData.State[1].MasterFactor		 := REAL_TO_UDINT((MatchedSpeed_Inch-rTempPosA1_Inch)*gA[11].UnitsPerInch);
				AutData.State[1].SlaveFactor		 := REAL_TO_UDINT((MatchedSpeed_Inch-rTempPosA1_Inch)*gA[1].UnitsPerInch);
				AutData.State[1].CompMode			   := ncOFF;

				AutData.State[1].Event[0].Type		  := ncST_END ;
				AutData.State[1].Event[0].Attribute	:= ncST_END;
				AutData.State[1].Event[0].NextState	:= 2;

			//Initial Comp With Matched Speed Zone
				AutData.State[2].CamProfileIndex  	:= 16#FFFF;
				AutData.State[2].MasterFactor		    := REAL_TO_UDINT(MatchedSpeed_Inch*gA[11].UnitsPerInch);
				AutData.State[2].SlaveFactor		    := REAL_TO_UDINT(MatchedSpeed_Inch*gA[1].UnitsPerInch);
				AutData.State[2].CompMode		    	  := ncONLYCOMP;
				AutData.State[2].MasterCompDistance	:= (gA[11].AxisPeriod)-((gA[11].PositionInch+MasterOffset)*gA[11].UnitsPerInch)-AutData.State[1].MasterFactor;
				AutData.State[2].SlaveCompDistance	:= (Slave_AxisPeriod)-gA[1].PositionCount-AutData.State[1].SlaveFactor;

				IF (AutData.State[2].SlaveCompDistance<=0) THEN
					AutData.State[2].SlaveCompDistance := AutData.State[2].SlaveCompDistance+Slave_AxisPeriod;
				END_IF
				IF (AutData.State[2].MasterCompDistance<0) THEN
					Value1 := REAL_TO_DINT(AutData.State[2].MasterCompDistance);
					Value2 := REAL_TO_DINT(gA[11].AxisPeriod);
					AutData.State[2].MasterCompDistance := DINT_TO_REAL(Value1 MOD Value2);
					IF (AutData.State[2].MasterCompDistance<0) THEN
						AutData.State[2].MasterCompDistance := AutData.State[2].MasterCompDistance+gA[11].AxisPeriod;
					END_IF
				END_IF

				IF ((AutData.State[2].MasterCompDistance<(0.5*gA[11].AxisPeriod)) AND (AutData.State[2].SlaveCompDistance>(0.5*Slave_AxisPeriod))) THEN
					AutData.State[2].MasterCompDistance := AutData.State[2].MasterCompDistance+(gA[11].AxisPeriod);
				END_IF

				AutData.State[2].Event[0].Type		:= ncST_END ;
				AutData.State[2].Event[0].Attribute	:= ncST_END;
				AutData.State[2].Event[0].NextState	:= 3;

			ELSE
				InMatched := 0;

			//Automat STATE 0 Basis State
				AutData.State[0].Event[0].Type		  := ncST_END;
				AutData.State[0].Event[0].Attribute	:= ncAT_ONCE;
				AutData.State[0].Event[0].NextState	:= 5;

			//Initial Comp With Matched Speed Zone
				AutData.State[5].CamProfileIndex := 16#FFFF;
				AutData.State[5].MasterFactor		 := REAL_TO_UDINT(MatchedSpeed_Inch*gA[11].UnitsPerInch);
				AutData.State[5].SlaveFactor		 := REAL_TO_UDINT(MatchedSpeed_Inch*gA[1].UnitsPerInch);
				AutData.State[5].CompMode			   := ncONLYCOMP;
				AutData.State[5].MasterCompDistance	:= gA[11].AxisPeriod-((gA[11].PositionInch+MasterOffset)*gA[11].UnitsPerInch);
				AutData.State[5].SlaveCompDistance	:= Slave_AxisPeriod-gA[1].PositionCount;

				IF (AutData.State[5].SlaveCompDistance<=0) THEN
					AutData.State[5].SlaveCompDistance := AutData.State[5].SlaveCompDistance+Slave_AxisPeriod;
				END_IF
				IF (AutData.State[5].MasterCompDistance<0) THEN
					Value1 := REAL_TO_DINT(AutData.State[5].MasterCompDistance);
					Value2 := REAL_TO_DINT(gA[11].AxisPeriod);
					AutData.State[5].MasterCompDistance := DINT_TO_REAL(Value1 MOD Value2);
					IF (AutData.State[5].MasterCompDistance<0) THEN
						AutData.State[5].MasterCompDistance := AutData.State[5].MasterCompDistance+gA[11].AxisPeriod;
					END_IF
				END_IF

				IF ((AutData.State[5].MasterCompDistance<(0.5*gA[11].AxisPeriod)) AND (AutData.State[5].SlaveCompDistance>(0.5*Slave_AxisPeriod))) THEN
					AutData.State[5].MasterCompDistance := AutData.State[5].MasterCompDistance+(gA[11].AxisPeriod);
				END_IF

				AutData.State[5].Event[0].Type		  := ncST_END ;
				AutData.State[5].Event[0].Attribute	:= ncST_END;
				AutData.State[5].Event[0].NextState	:= 3;

			END_IF

    //Running Comp With Matched Speed Zone
      AutData.State[3].CamProfileIndex    := 16#FFFF;
      AutData.State[3].MasterFactor       := REAL_TO_UDINT(MatchedSpeed_Inch*gA[11].UnitsPerInch);
      AutData.State[3].SlaveFactor        := REAL_TO_UDINT(MatchedSpeed_Inch*gA[1].UnitsPerInch);
      AutData.State[3].CompMode           := ncONLYCOMP;
      AutData.State[3].MasterCompDistance := gA[11].AxisPeriod-AutData.State[3].MasterFactor;
      AutData.State[3].SlaveCompDistance  := Slave_AxisPeriod-AutData.State[3].SlaveFactor;

      AutData.State[3].Event[0].Type      := ncST_END ;
      AutData.State[3].Event[0].Attribute := ncST_END;
      AutData.State[3].Event[0].NextState := 3;

		//Initialize & Enable the Automat Control
			MC_BR_AutControl_0.Enable 		:= 1;
			MC_BR_AutControl_0.AdrAutData 	:= ADR(AutData);
			MC_BR_AutControl_0.InitAutData 	:= 1;
	END_IF
		// wait for initialization done
			IF ((MC_BR_AutControl_0.AutDataInitialized = 1) AND (Synch_Request)) THEN
				MC_BR_AutControl_0.InitAutData 	:= 0;
				AutomatStart := 1;
			END_IF
			// check if error occured
			IF (MC_BR_AutControl_0.ErrorID <> 0) THEN
				MC_BR_AutControl_0.Enable := 0;
				uiErrorID := MC_BR_AutControl_0.ErrorID ;
			END_IF

	(******************** ENABLE CAM-AUTOMAT **********************)

	IF (AutomatStart) THEN
			MC_BR_AutControl_0.Start := 1;
			AutomatStart := 0;
	END_IF

  IF (NOT Synch_Request) THEN
			MC_BR_AutControl_0.Stop := 1;
			MC_BR_AutControl_0.Start := 0;
			ParID_Ready := 0;
			IF (MC_BR_AutControl_0.Running=0) THEN
				MC_BR_AutControl_0.Enable := 0;
				MC_BR_AutControl_0.Stop := 0;
			END_IF
	END_IF

	IF (NOT gPerf_ParkRequired) THEN
		gA[1].Ind_AutomatEnabled:=MC_BR_AutControl_0.Enable;
		gA[1].Ind_CurrentAutomatState:=MC_BR_AutControl_0.ActualStateIndex;
	END_IF
  gA[1].Ind_bSynchroOK := (MC_BR_AutControl_0.ActualStateIndex >= 2) AND gA[1].Ind_SynchronizedMotion ;
	(********************** MC_AUTCONTROL *************************)
	MC_BR_AutControl_0.Slave:= gA[1].Ident;
	MC_BR_AutControl_0();

	(******************** UPDATE CAM-AUTOMAT STATE 3 **********************)
	MC_BR_InitAutState_0.Master := gA[11].Ident;
	MC_BR_InitAutState_0.Slave := gA[1].Ident;
	MC_BR_InitAutState_0.StateIndex := 3;
	MC_BR_InitAutState_0.CamProfileIndex := 16#FFFF;
	MC_BR_InitAutState_0.MasterFactor := REAL_TO_UDINT(MatchedSpeed_Inch*gA[11].UnitsPerInch);
	MC_BR_InitAutState_0.SlaveFactor := REAL_TO_UDINT(MatchedSpeed_Inch*gA[1].UnitsPerInch);
	MC_BR_InitAutState_0.MasterCompDistance := gA[11].AxisPeriod-MC_BR_InitAutState_0.MasterFactor;
	MC_BR_InitAutState_0.SlaveCompDistance	:= Slave_AxisPeriod-MC_BR_InitAutState_0.SlaveFactor;
	MC_BR_InitAutState_0.Execute := gA[1].Cmd_SynchronizedMotionUpdate;
	MC_BR_InitAutState_0();

  IF (MC_BR_InitAutState_0.Done OR MC_BR_InitAutState_0.Error) THEN
		gA[1].Cmd_SynchronizedMotionUpdate:=0;
	END_IF

END_PROGRAM
```

#### A1_Automat.var - Local variables
```iecst
(********************************************************************
 * COPYRIGHT -- Microsoft
 ********************************************************************
 * Program: A1_Automat
 * File: A1_Automat.var
 * Author: pkiel
 * Created: July 12, 2011
 ********************************************************************
 * Local variables of program A1_Automat
 ********************************************************************)
VAR
	AutData : MC_AUTDATA_TYP;
	AutomatStart : BOOL;
	ErrorID : UINT;
	InMatched : BOOL;
	MasterOffset : REAL;
	MasterParID : UINT;
	MatchedSpeed_Inch : REAL;
	MC_BR_AutControl_0 : MC_BR_AutControl;
	MC_BR_InitAutState_0 : MC_BR_InitAutState;
	MC_BR_InitMasterParIDTransfer_0 : MC_BR_InitMasterParIDTransfer;
	ParID_Ready : BOOL;
	PositionMOD : DINT;
	PositionOffset : DINT;
	Slave_AxisPeriod : REAL;
	rSlave_AxisPeriod_Inch : REAL;
	rPosOutMatchedSpeed2_Inch : REAL;
	SlaveStartOffset : REAL;
	Synch_Request : BOOL;
	Value1 : DINT;
	Value2 : DINT;
	bTest_ : ARRAY[0..9] OF BOOL;
	rPhaseTest : REAL;
	bInitCamAuto : BOOL;
	bCalcCameProf : BOOL;
	uiErrorID : UINT := 0;
	bTest : BOOL;
	rTest_ : ARRAY[0..9] OF REAL ;
	rTempPosA1_Inch : REAL;
END_VAR
```

### Program Logical/BagMachine_Section/Perf/Axis1/A1_Automat2 (IEC)

#### A1_Automat2.var - Local variables
```iecst
(********************************************************************
 * COPYRIGHT -- Microsoft
 ********************************************************************
 * Program: A1_Automat2
 * File: A1_Automat2.var
 * Author: pkiel
 * Created: July 19, 2011
 ********************************************************************
 * Local variables of program A1_Automat2
 ********************************************************************)
VAR
  AutData : MC_AUTDATA_TYP;
  AutomatStart : BOOL;
  Error : UINT;
  ErrorID : UINT;
  InMatched : BOOL;
  MasterOffset : REAL;
  MasterParID : UINT;
  MatchedSpeed_Inch : REAL;
  MC_BR_AutControl_0 : MC_BR_AutControl;
  MC_BR_InitMasterParIDTransfer_0 : MC_BR_InitMasterParIDTransfer;
  ParID_Ready : BOOL;
  Slave_AxisPeriod : REAL;
  SlaveTravel_Deg : REAL;
  Synch_Request : BOOL;
  Travel_Deg : REAL;
  Travel_Inch : REAL;
  Value1 : DINT;
  Value2 : DINT;
  rSlave_AxisPeriod_Inch : REAL ;
  rPosOutMatchedSpeed2_Inch : REAL;
  rTempPosA1_Inch : REAL ;
  bInitCamAuto : BOOL ;

END_VAR
```

### Program Logical/BagMachine_Section/Perf/Axis1/A1_Basic (IEC)

#### A1_BasicCyclic.st - Cyclic code
```iecst
(********************************************************************
 * COPYRIGHT -- Microsoft
 ********************************************************************
 * Program: A1_Basic
 * File: A1_BasicCyclic.st
 * Author: pkiel
 * Created: July 11, 2011
 ********************************************************************
 * Implementation of program A1_Basic
 ********************************************************************)

PROGRAM _CYCLIC

	IF (gA[1].Ident<>0) THEN

	(************************ READ DRIVE STATUS *************************)
	(* Access to the following bools:
	gA[x]_DriveStatus.Simulation			: If TRUE, simulation mode is active
	gA[x]_DriveStatus.NetworkInit			: If TRUE, the network is initialized
	gA[x]_DriveStatus.HomeSwitch			: If TRUE, the digital reference switch input is active
	gA[x]_DriveStatus.PosHWSwitch			: If TRUE, the positive hardware end switch is active
	gA[x]_DriveStatus.NegHWSwitch			: If TRUE, the negative hardware end switch is active
	gA[x]_DriveStatus.Trigger1				: If TRUE, the first trigger input is active
	gA[x]_DriveStatus.Trigger2				: If TRUE, the second trigger input is active
	gA[x]_DriveStatus.DriveEnable			: If TRUE, the enable input is active
	gA[x]_DriveStatus.ControllerReady		: If TRUE, the controller is ready to beturned on
	gA[x]_DriveStatus.ControllerStatus		: If TRUE, the controller is turned on (Same as MC_Power.Status)
	gA[x]_DriveStatus.AxisError				: If TRUE, at least one error has occurred (not acknowledged)
	gA[x]_DriveStatus.LagWarning			: If TRUE, the lag error has exceeded the limit value specified for a warning*)
		MC_BR_ReadDriveStatus_0.Enable := 1;
		MC_BR_ReadDriveStatus_0.Axis := gA[1].Ident;
		MC_BR_ReadDriveStatus_0.AdrDriveStatus := ADR (DriveStatus);
		MC_BR_ReadDriveStatus_0();
		gA[1].Ind_Simulation		:=	DriveStatus.Simulation;
		gA[1].Ind_NetworkInit		:=	DriveStatus.NetworkInit;
		gA[1].Input_Home			:=	DriveStatus.HomeSwitch;
		gA[1].Input_PosHW			:=	DriveStatus.PosHWSwitch;
		gA[1].Input_NegHW			:=	DriveStatus.NegHWSwitch;
		gA[1].Input_Trigger1		:=	DriveStatus.Trigger1;
		gA[1].Input_Trigger2		:=	DriveStatus.Trigger2;
		gA[1].Input_DriveEnable		:=	DriveStatus.DriveEnable;
		gA[1].Ind_ControllerReady	:=	DriveStatus.ControllerReady;
		gA[1].Ind_ControllerStatus	:=	DriveStatus.ControllerStatus;
		gA[1].Error					:=	DriveStatus.AxisError;
		gA[1].Ind_LagWarning		:=	DriveStatus.LagWarning;

	(************************ READ AXIS ERROR **********************)
		MC_ReadAxisError_0.Enable := gA[1].Ind_NetworkInit;
		MC_ReadAxisError_0.Axis := gA[1].Ident;
		MC_ReadAxisError_0.DataAddress := ADR(gA[1].ErrorText);
		MC_ReadAxisError_0.DataLength := SIZEOF(gA[1].ErrorText);
		MC_ReadAxisError_0.DataObjectName := 'Error_Eng';
		MC_ReadAxisError_0();
		IF(MC_ReadAxisError_0.Valid) THEN
			gA[1].ErrorID := MC_ReadAxisError_0.AxisErrorID;
			gA[1].ErrorCount := MC_ReadAxisError_0.AxisErrorCount;
		END_IF
	(* Auto Acknowledge Errors *)
		IF (gA[1].Cmd_Reset AND (gA[1].ErrorCount<>0) AND NOT AutoAck) THEN
			AutoAck:=1;
		ELSE
			AutoAck:=0;
		END_IF
	(*Axis Error Acknowledge*)
		IF (EDGEPOS(AutoAck) OR EDGEPOS(gA[1].ErrorAck)) THEN
			MC_ReadAxisError_0.Acknowledge := 1;
		ELSE;
			MC_ReadAxisError_0.Acknowledge :=0;
		END_IF

	(************************ RESET AXIS ERROR **********************)
		IF (gA[1].Cmd_Reset AND (gA[1].ErrorCount=0) AND gA[1].ErrorStop) THEN
			MC_Reset_0.Execute:=1;
		END_IF
		IF (MC_Reset_0.Done) THEN
			MC_Reset_0.Execute:=0;
			gA[1].Cmd_Reset:=0;
			ResetError := 0;
		END_IF
		IF (MC_Reset_0.Error) THEN
			MC_Reset_0.Execute:=0;
			gA[1].Cmd_Reset:=0;
			ResetError := 1;
		END_IF
		MC_Reset_0.Axis:=gA[1].Ident;
		MC_Reset_0();

	(************************ READ AXIS STATUS *************************)
		MC_ReadStatus_0.Enable := gA[1].Ind_NetworkInit;
		MC_ReadStatus_0.Axis := gA[1].Ident;
		MC_ReadStatus_0();
		IF(MC_ReadStatus_0.Valid = TRUE)THEN
			gA[1].Ind_Enabled 			:= NOT (MC_ReadStatus_0.Disabled);
			gA[1].Ind_StandStill		:= MC_ReadStatus_0.StandStill;
			gA[1].Ind_Stopping			:= MC_ReadStatus_0.Stopping;
			gA[1].Ind_DiscreteMotion	:= MC_ReadStatus_0.DiscreteMotion;
			gA[1].Ind_ContinuousMotion	:= MC_ReadStatus_0.ContinuousMotion;
			gA[1].Ind_SynchronizedMotion:= MC_ReadStatus_0.SynchronizedMotion;
			gA[1].ErrorStop				:= MC_ReadStatus_0.Errorstop;
    END_IF
    IF NOT(gA[1].Ind_Enabled) THEN
      gA[1].bSynchroReq := 1 ;
    END_IF
    IF EDGEPOS(gA[1].Ind_bSynchroOK) THEN
      gA[1].bSynchroReq := 0 ;
    END_IF

	(******************** INIT POSITION MODULUS  *********************)
		MC_BR_InitModPos_0.Execute:= InitModPosition;
		MC_BR_InitModPos_0.Axis:= gA[1].Ident;
		MC_BR_InitModPos_0.Period:= REAL_TO_UDINT(gA[1].AxisPeriod);
		MC_BR_InitModPos_0.Factor:=1;
		InitModPos_Done:=MC_BR_InitModPos_0.Done;
		MC_BR_InitModPos_0();

	(******************** INIT ENDLESS POSITION *********************)
		MC_BR_InitEndlessPosition_0.Execute:= InitModPos_Done;
		MC_BR_InitEndlessPosition_0.Axis:= gA[1].Ident;
		MC_BR_InitEndlessPosition_0.DataAddress:= ADR(gEndPosData[1]);
		IF (MC_BR_InitEndlessPosition_0.Done) THEN
			InitModPosition:=0;
			InitEndlessPosition:=0;
			HomeRestore:=1;
		END_IF
		MC_BR_InitEndlessPosition_0();

	(************************ HOME AXIS FIRST POWER UP **********************)
		IF (HomeRestore AND NOT gA1_FirstHomed) THEN
			MC_Home_0.Execute:=1;
		END_IF
		MC_Home_0.Axis:=gA[1].Ident;
		MC_Home_0.Position:=0;
		MC_Home_0.HomingMode:=mcHOME_DIRECT;
		IF (MC_Home_0.Done) THEN
			MC_Home_0.Execute:=0;
			gA1_FirstHomed:=1;
		END_IF
		MC_Home_0();

	(************************ HOME AXIS **********************)
		IF (gA1_FirstHomed) THEN
			MC_Home_1.Execute:=HomeRestore;
		END_IF
		MC_Home_1.Axis:=gA[1].Ident;
		MC_Home_1.Position:=0;
		MC_Home_1.HomingMode:=mcHOME_RESTORE_POS;
		IF (MC_Home_1.Done) THEN
			gA[1].Ind_Homed:=1;
			HomeRestore:=0;
		END_IF
		MC_Home_1();

  (******************** READ ACTUAL POSITION *********************)
    MC_ReadActualPosition_0.Enable:= gA[1].Ind_NetworkInit;
    MC_ReadActualPosition_0.Axis:= gA[1].Ident;
    MC_ReadActualPosition_0();
    IF(MC_ReadActualPosition_0.Valid = TRUE)THEN
      gA[1].PositionCount := MC_ReadActualPosition_0.Position;
      gA[1].PositionInch := gA[1].PositionCount/gA[1].UnitsPerInch;
      gA[1].PositionDeg := gA[1].PositionCount/gA[1].UnitsPerDeg;
    END_IF

  //******************** REVOLUTION COUNT *********************
    IF EDGEPOS(gA[1].PositionDeg > 60.0) THEN
      IF gA[1].uiiNumRev = 4294967295 THEN
        gA[1].uiiNumRev := 1 ;
      ELSE
        gA[1].uiiNumRev := gA[1].uiiNumRev + 1 ;
      END_IF
    END_IF

  //******************** READ SET POINT POSITION *********************
    // Slave side  : ParID 428 SGEN_S_SET : CTRL Position controller: Input set position
    // Master side : ParID 412 S_SET_VAX1 : 412: VAX: Position

    // Slave side
    MC_BR_CyclicRead_0.Axis        := gA[11].Ident ; //gA[1].Ident ;
    MC_BR_CyclicRead_0.Enable      := gA[1].Ind_NetworkInit;
    MC_BR_CyclicRead_0.ParID       := 412 ; //428 ;
    MC_BR_CyclicRead_0.DataAddress := ADR(iiSP_SlPos_U);
    MC_BR_CyclicRead_0.DataType    := ncPAR_TYP_DINT ;
    // Master side
    MC_BR_CyclicRead_1.Axis        := gA[9].Ident ;
    MC_BR_CyclicRead_1.Enable      := gA[1].Ind_NetworkInit;
    MC_BR_CyclicRead_1.ParID       := 412 ;
    MC_BR_CyclicRead_1.DataAddress := ADR(iiSP_MaPos_U);
    MC_BR_CyclicRead_1.DataType    := ncPAR_TYP_DINT ;

    IF MC_BR_CyclicRead_0.Valid THEN
      //rSP_SlPos_Deg := REAL_TO_UDINT((iiSP_SlPos_U/gA[1].UnitsPerDeg)) MOD 360/gSP_PerfKnifeCount ;
      rSP_SlPos_Deg := iiSP_SlPos_U/gA[1].UnitsPerDeg ;
    ELSIF MC_BR_CyclicRead_0.Error THEN
      MC_BR_CyclicRead_0.Enable := 0 ;
    END_IF
    IF MC_BR_CyclicRead_1.Valid THEN
      //rSP_MaPos_Deg := REAL_TO_UDINT((iiSP_MaPos_U/gA[9].UnitsPerDeg)) MOD 360 ;
      rSP_MaPos_Deg := iiSP_MaPos_U/gA[9].UnitsPerDeg ;
    ELSIF MC_BR_CyclicRead_1.Error THEN
      MC_BR_CyclicRead_1.Enable := 0 ;
    END_IF
    MC_BR_CyclicRead_0();
    MC_BR_CyclicRead_1();

  //******************** READ ACTUAL OFFSET *********************
  rTempPosA1_Deg := H_FC_Modulus(IN_rMod:=360/gSP_PerfKnifeCount, IN_rVar:=gA[1].PositionDeg) ;
  g_bPerfInMatchedSpeed := ( rTempPosA1_Deg < gSP_A[1].MatchedSpeed ) ;
  IF //g_bPerfInMatchedSpeed      AND
     g_rActualSizePerf_in > 0.0 THEN
    //rTempActPhasDeg := rSP_SlPos_Deg - gRecipeActive.Repeat/g_rActualSizePerf_in * rSP_MaPos_Deg ;
    rTempActPhasDeg := rSP_SlPos_Deg - rSP_MaPos_Deg ;
    gA[1].rActPhasDeg := H_FC_Modulus (
                              IN_rMod := 360,
                              IN_rVar := rTempActPhasDeg
                                      ) ;
  END_IF

	(******************** READ ACTUAL VELOCITY *********************)
		IF(MC_ReadActualVelocity_0.Error=TRUE) THEN
			MC_ReadActualVelocity_0.Enable:= 0;
		ELSE
			MC_ReadActualVelocity_0.Enable:= 1;
		END_IF
		MC_ReadActualVelocity_0.Axis:= gA[1].Ident;
		MC_ReadActualVelocity_0();
		IF(MC_ReadActualVelocity_0.Valid = TRUE)THEN
			//gA[1].ActualVelocity := MC_ReadActualVelocity_0.Velocity*60/gA[1].SP_MotorPPR;
      gA[1].ActualVelocity := MC_ReadActualVelocity_0.Velocity*60/gA[1].AxisPeriod ; // D.M. 03/08/2011 BrownPaper_14542  Need speed of the axis and not of the shaft of the motor
      IF (ABS(gA[1].ActualVelocity)>1) THEN // D.M. 03/08/2011 BrownPaper_14542 Add ABS because in case negative velocity Ind_InMotion = 0 instead of 1
				gA[1].Ind_InMotion:=1;
			ELSE
				gA[1].Ind_InMotion:=0;
			END_IF
		END_IF

	(******************** READ ACTUAL TORQUE *********************)
		IF(MC_ReadActualTorque_0.Error=TRUE) THEN
			MC_ReadActualTorque_0.Enable:= 0;
		ELSE
			MC_ReadActualTorque_0.Enable:= 1;
		END_IF
		MC_ReadActualTorque_0.Axis:= gA[1].Ident;
		MC_ReadActualTorque_0();
		IF(MC_ReadActualTorque_0.Valid = TRUE)THEN
			gA[1].ActualTorque := MC_ReadActualTorque_0.Torque;
		END_IF

	(************************ ENABLE AXIS **********************)
		MC_Power_0.Axis:=gA[1].Ident;
		IF (MC_Power_0.Error=0) THEN
			MC_Power_0.Enable:=gA[1].Cmd_Enable;
		ELSE;
			MC_Power_0.Enable:=0;
		END_IF;
		MC_Power_0();

	(************************ AXIS VELOCITY MOVE **********************)
    IF (((EDGEPOS(gA[1].Cmd_ContinuousMotion)) OR (EDGEPOS(gA[1].Cmd_ContinuousMotionUpdate)))) THEN
			MC_MoveVelocity_0.Execute:=1;
      rAxisTimSet_SP_Vel  := gA[1].SP_Velocity*gA[1].AxisPeriod/60;
      rAxisTimSet_SP_Acc  := gA[1].SP_Accel;
      rAxisTimSet_SP_Dec  := gA[1].SP_Decel;
      uiAxisTimSet_SP_Dir := mcPOSITIVE_DIR;
    ELSIF gstCycA[1].CycManTimSet.CmdMov AND 0 THEN
      MC_MoveVelocity_0.Execute := 1 ;
      rAxisTimSet_SP_Vel := gr_rAxisTimSet_SP_Vel*gA[1].AxisPeriod/60 ;
      rAxisTimSet_SP_Acc := gr_rAxisTimSet_SP_Acc*gA[1].AxisPeriod/60/60 ;
      rAxisTimSet_SP_Dec := gr_rAxisTimSet_SP_Dec*gA[1].AxisPeriod/60/60 ;
      IF gA[1].Cmd_ManuTimSetPlus THEN
        uiAxisTimSet_SP_Dir := mcPOSITIVE_DIR;
      ELSE
        uiAxisTimSet_SP_Dir := mcNEGATIVE_DIR;
      END_IF;
		ELSE
			MC_MoveVelocity_0.Execute:=0;
		END_IF;
    MC_MoveVelocity_0.Axis         := gA[1].Ident ;
    MC_MoveVelocity_0.Velocity     := rAxisTimSet_SP_Vel ;
    MC_MoveVelocity_0.Acceleration := rAxisTimSet_SP_Acc ;
    MC_MoveVelocity_0.Deceleration := rAxisTimSet_SP_Dec ;
    MC_MoveVelocity_0.Direction    := uiAxisTimSet_SP_Dir ;
	MC_MoveVelocity_0();

  //************************ AXIS OVERRIDE **********************
    MC_SetOverride_0.Axis      := gA[1].Ident ;
    MC_SetOverride_0.Enable    := gA[1].Cmd_Override ;
    MC_SetOverride_0.VelFactor := gA[1].rSP_OverrideV ;
    MC_SetOverride_0.AccFactor := gA[1].rSP_OverrideA ;
    IF (MC_SetOverride_0.Enabled) OR
       (MC_SetOverride_0.Error)   THEN
      gA[1].Cmd_Override := 0 ;
    END_IF
    MC_SetOverride_0();

	(************************ AXIS STOP **********************)
		MC_Stop_0.Axis:=gA[1].Ident;
    IF (gA[1].Ind_ContinuousMotion AND (NOT gA[1].Cmd_ContinuousMotion) AND gAlarmsOK) THEN
			MC_Stop_0.Deceleration:=gA[1].SP_Decel;
			MC_Stop_0.Execute:=1;
		END_IF;
		IF (MC_Stop_0.Done OR MC_Stop_0.CommandAborted OR MC_Stop_0.Error) THEN
			MC_Stop_0.Execute:=0;
		END_IF;
		MC_Stop_0();

  (************************  ESTOP **********************)
    MC_Stop_1.Axis:=gA[1].Ident;
    IF EDGEPOS(g_bIndEStopStandstill) THEN
      MC_Stop_1.Deceleration:=gA[1].SP_EStopDecel;
      MC_Stop_1.Execute:=1;
    END_IF;
    IF (MC_Stop_1.Done OR MC_Stop_1.CommandAborted OR MC_Stop_1.Error) THEN
      MC_Stop_1.Execute:=0;
      gA[1].Cmd_EStopDisable := 1 ;
    END_IF;
    IF NOT(g_bIndEStopStandstill) THEN
      gA[1].Cmd_EStopDisable := 0 ;
    END_IF;
    MC_Stop_1();

		(************************ AXIS PHASE CONTROL (Inches) **********************)
		(*MC_BR_Phasing_0.Slave:=gA[1].Ident;
    IF (gA[1].Ind_SynchronizedMotion) THEN
			MC_BR_Phasing_0.Enable:=1;
		ELSE
			MC_BR_Phasing_0.Enable:=0;
		END_IF;
    IF (gA[1].Cmd_PhaseOffset) THEN
			MC_BR_Phasing_0.InitData:=1;
			gA[1].Cmd_PhaseOffset:=0;
    ELSE
			MC_BR_Phasing_0.InitData:=0;
		END_IF ;

		(*IF(gA[9].Ind_InMotion) THEN
			MC_BR_Phasing_0.ApplicationMode:=mcMASTER_DISTANCE_BASED;
		ELSE*)
		(*END_IF*)
		MC_BR_Phasing_0.Shift:=gA[1].SP_PhaseOffset*gA[9].UnitsPerInch ;
		MC_BR_Phasing_0.Velocity            := rAxisTimSet_SP_Vel;
		MC_BR_Phasing_0.Acceleration        := rAxisTimSet_SP_Acc;
		MC_BR_Phasing_0.ApplicationDistance := 2*gA[9].AxisPeriod;
		MC_BR_Phasing_0.ShiftMode           := mcRELATIVE;
    MC_BR_Phasing_0.ApplicationMode     := uiAxisTimSet_SP_ShiftAppMode;
    MC_BR_Phasing_0.PerformVelocityControl := gstCycA[1].CycManTimSet.CmdMov AND 0 ;
		MC_BR_Phasing_0();

	END_IF

END_PROGRAM
```
